(* Logix 5000 project; controller HP_SSC01 vendor 1 type 14 code 67 rev 17.7; software revision 17.01 *)

TASK MainTask (periodic, rate 10 ms, priority 5, watchdog 50 ms) : Main_SSC, Carousel1, Carousel2
TASK SafetyTask (periodic, rate 25 ms, priority 10, watchdog 20 ms) : Safe_SSC, SafeCarousel1

MODULES
   Local : vendor 1 type 14 code 67 (ICP 0, rev 17.7)
      SSC01_DNetSafeIO : vendor 1 type 12 code 14 (ICP 5, rev 10.5, Output RPI 20 ms, Input RPI 20 ms)
         SSC01_Safe2 : vendor 1 type 35 code 2 (DeviceNet 2, rev 1.2, Output RPI 25 ms, Input RPI 6 ms)
         C2_Safe : vendor 1 type 35 code 2 (DeviceNet 20, rev 1.2, Output RPI 25 ms, Input RPI 6 ms)
         SSC01_Safe3 : vendor 1 type 35 code 2 (DeviceNet 3, rev 1.2, Output RPI 25 ms, Input RPI 6 ms)
         C3_Safe : vendor 1 type 35 code 2 (DeviceNet 30, rev 1.2, Output RPI 25 ms, Input RPI 6 ms)
         SSC01_Safe1 : vendor 1 type 35 code 2 (DeviceNet 1, rev 1.2, Output RPI 25 ms, Input RPI 6 ms)
         C1_Safe : vendor 1 type 35 code 2 (DeviceNet 10, rev 1.2, Input RPI 6 ms, Output RPI 25 ms)
      HP_SSC01_0_3_ENBT : 1756-ENBT (ICP 3, Ethernet 192.168.201.51, rev 4.1)
         HP_RCS_RIDE_ENBT : 1756-ENBT (Ethernet 192.168.201.10, rev 4.1)
            @fd516503@:Partner : vendor 1 type 14 code 69 (ICP 1, rev 16.1)
            HP_RCS : vendor 1 type 14 code 67 (ICP 0, rev 16.1, $55e8e5d5$ RPI 25 ms)
      HP_SSC01_0_6_EN2T : 1756-EN2T (ICP 6, Ethernet 192.168.206.10, rev 1.3)
         C2_RIO_AENT : 1734-AENT (Ethernet 192.168.206.21, rev 2.3, Output RPI 20 ms)
            C2_RIO_1_IB8 : 1734-IB8 (PointIO 1, rev 3.1)
            C2_RIO_2_OB8 : 1734-OB8 (PointIO 2, rev 3.1)
            C2_RIO_3_SSI : vendor 1 type 115 code 80 (PointIO 3, rev 4.3, Output RPI 10 ms)
         C1_RIO_AENT : 1734-AENT (Ethernet 192.168.206.11, rev 2.3, Output RPI 20 ms)
            C1_RIO_1_IB8 : 1734-IB8 (PointIO 1, rev 3.1)
            C1_RIO_2_OB8 : 1734-OB8 (PointIO 2, rev 3.1)
            C1_RIO_3_SSI : vendor 1 type 115 code 80 (PointIO 3, rev 4.3, Output RPI 10 ms)
         C3_RIO_AENT : 1734-AENT (Ethernet 192.168.206.31, rev 2.3, Output RPI 20 ms)
            C3_RIO_1_IB8 : 1734-IB8 (PointIO 1, rev 3.1)
            C3_RIO_3_SSI : vendor 1 type 115 code 80 (PointIO 3, rev 4.3, Output RPI 10 ms)
            C3_RIO_2_OB8 : 1734-OB8 (PointIO 2, rev 3.1)
      HP_SSC01_0_2_ENBT : 1756-ENBT (ICP 2, Ethernet 192.168.202.11, rev 4.1)
      C1_SERCOS : vendor 1 type 16 code 13 (ICP 8, rev 17.1, MotionSync RPI 6 ms, MotionAsync RPI 25 ms, MotionEvent RPI 1000 ms)
         C1_K7K : vendor 1 type 115 code 182 (SERCOS 1, rev 1.1)
      C3_SERCOS : vendor 1 type 16 code 13 (ICP 10, rev 17.1, MotionSync RPI 6 ms, MotionAsync RPI 25 ms, MotionEvent RPI 1000 ms)
         C3_K7K : vendor 1 type 115 code 182 (SERCOS 3, rev 1.1)
      C2_SERCOS : vendor 1 type 16 code 13 (ICP 9, rev 17.1, MotionSync RPI 6 ms, MotionAsync RPI 25 ms, MotionEvent RPI 1000 ms)
         C2_K7K : vendor 1 type 115 code 182 (SERCOS 2, rev 1.1)
      @b5ff5b04@:Partner : vendor 1 type 14 code 69 (ICP 1, rev 17.7)
END_MODULES

TYPE FAULTRECORD :
STRUCT
   Time_Low : DINT;
   Time_High : DINT;
   Type : INT;
   Code : INT;
   Info : DINT[8];
END_STRUCT
END_TYPE

TYPE Profile_Table_Limits :
STRUCT
   On_Path_Low : REAL;
   On_Path_High : REAL;
   Near_On_Path_Low : REAL;
   Near_On_Path_High : REAL;
END_STRUCT
END_TYPE

TYPE UD_DTS :
STRUCT
   YEAR : DINT;
   MONTH : DINT;
   DAY : DINT;
   HOUR : DINT;
   MINUTE : DINT;
   SECOND : DINT;
   MIL_SEC : DINT;
END_STRUCT
END_TYPE

TYPE UD_FH_DATA :
STRUCT
   CODE : INT;
   MESSAGE : DINT;
   DATE_TIME : UD_DTS;
END_STRUCT
END_TYPE

TYPE UD_FH_LOG :
STRUCT
   MESSAGE : DINT;
   YEAR : DINT;
   MONTH : DINT;
   DAY : DINT;
   HOUR : DINT;
   MINUTE : DINT;
   SECOND : DINT;
   MIL_SEC : DINT;
END_STRUCT
END_TYPE

TYPE Udt_Carsl_SafeData :
STRUCT
   Status : CONNECTION_STATUS;
   Carsl_Status : DINT;
END_STRUCT
END_TYPE

TYPE Udt_Carsl_Stat :
STRUCT
   Enabled : BOOL;
   Mode : UDT_MODE;
   Posn : UDT_PositionProfile;
   Position : UDT_Parameter_Delta;
   CogNo : REAL;
   CogPosition : REAL;
   Velocity : REAL;
   PosnStatus : UDT_Position_Status;
   MotionCmdEn : BOOL;
   MotionActive : BOOL;
   realCog : REAL;
   realCogTot : REAL;
   RevCount : COUNTER;
   RevFlag : BOOL;
   Encoder_Secnd_Posn : REAL;
END_STRUCT
END_TYPE

TYPE UDT_Cog_Posn :
STRUCT
   CogNo : DINT;
   CogPosition : DINT;
   realCog : DINT;
   modCog : DINT;
END_STRUCT
END_TYPE

TYPE UDT_Encoder :
STRUCT
   Position : DINT;
   CntRaw : DINT;
   CntAdj : DINT;
   Initial : DINT;
   Delta : DINT;
   InitialPrev : DINT;
   CntMax : DINT;
   Rollover : DINT;
END_STRUCT
END_TYPE

TYPE UDT_GLX_ProduceConsume :
STRUCT
   Status : CONNECTION_STATUS;
   Data : DINT[5];
END_STRUCT
END_TYPE

TYPE UDT_MODE :
STRUCT
   Local : BOOL;
   Off : BOOL;
   Remote : BOOL;
   Unknown : BOOL;
END_STRUCT
END_TYPE

TYPE UDT_MOTION_STATE :
STRUCT
   Accel : BOOL;
   Run : BOOL;
   Decel : BOOL;
   Off : BOOL;
   OS : BOOL;
END_STRUCT
END_TYPE

TYPE UDT_Parameter_Delta :
STRUCT
   CurrentAbs : REAL;
   Initial : REAL;
   CurrentRel : REAL;
   Delta : REAL;
   Final : REAL;
END_STRUCT
END_TYPE

TYPE UDT_ParameterDint_Delta :
STRUCT
   Current : DINT;
   Initial : DINT;
   CurrentRel : DINT;
   Delta : DINT;
   Final : DINT;
END_STRUCT
END_TYPE

TYPE UDT_Position_Status :
STRUCT
   OnPath : BOOL;
   NearOnPath : BOOL;
   OffPath : BOOL;
   RecoveryZn : BOOL;
END_STRUCT
END_TYPE

TYPE UDT_PositionProfile :
STRUCT
   Initial : REAL;
   Accel : REAL;
   Stop : REAL;
   Final : REAL;
END_STRUCT
END_TYPE

TYPE Udt_RCS_SafeData :
STRUCT
   Status : CONNECTION_STATUS;
   Master_Clock : DINT;
   cst_Msec : DINT;
   cst_Sec : DINT;
   RailStateEthernet : DINT;
   Permissives : DINT;
END_STRUCT
END_TYPE

TYPE Udt_RCS_State :
STRUCT
   Value : DINT;
   Maint : BOOL;
   Add_Veh : BOOL;
   Second_Park : BOOL;
   Spare : BOOL;
   Stn_Park : BOOL;
   Reset_Flt : BOOL;
   Rem_Veh : BOOL;
   Go_Evac : BOOL;
   Inspect : BOOL;
   Inspect_Reset : BOOL;
   Retract_SAE : BOOL;
   Brake_Test : BOOL;
   Go_Keyhole : BOOL;
   Acq_MClock : BOOL;
   Go_MClock : BOOL;
   Inspect_Done : BOOL;
   StartUp_Keyhole : BOOL;
   Pri_Restart : BOOL;
   Stn_Evac : BOOL;
   Auto_Run : BOOL;
   Unknown : BOOL;
END_STRUCT
END_TYPE

TYPE UDT_Seqn :
STRUCT
   En : BOOL;
   OS : BOOL;
   Dn : BOOL;
   Flt : BOOL;
   Step : DINT;
   Tmr : TIMER;
END_STRUCT
END_TYPE

TYPE UDT_Test_Record :
STRUCT
   StartPosn : REAL;
   EndPosn : REAL;
   EndDist : REAL;
   TestTime : DINT;
   AccelPosn : REAL;
   AccelTime : DINT;
   AccelDist : REAL;
   AccelErrorHi : REAL;
   AccelErrorLo : REAL;
   RunPosn : REAL;
   RunTime : DINT;
   RunDist : REAL;
   RunErrorHi : REAL;
   RunErrorLo : REAL;
   DecelPosn : REAL;
   DecelTime : DINT;
   DecelDist : REAL;
   DecelErrorHi : REAL;
   DecelErrorLo : REAL;
END_STRUCT
END_TYPE

VAR_GLOBAL   (* controller tags *)
   A_C1_0200 : ALIAS FOR S_C1_FaultSafety.0;
   A_C1_0201 : ALIAS FOR S_C1_FaultSafety.1;
   A_C1_0202 : ALIAS FOR S_C1_FaultSafety.2;
   A_C1_0203 : ALIAS FOR S_C1_FaultSafety.3;
   A_C1_0204 : ALIAS FOR S_C1_FaultSafety.4;
   A_C1_0205 : ALIAS FOR S_C1_FaultSafety.5;
   A_C1_0206 : ALIAS FOR S_C1_FaultSafety.6;
   A_C1_0207 : ALIAS FOR S_C1_FaultSafety.7;
   A_C1_0208 : ALIAS FOR S_C1_FaultSafety.8;
   A_C1_0209 : ALIAS FOR S_C1_FaultSafety.9;
   A_C1_0210 : ALIAS FOR S_C1_FaultSafety.10;
   A_C1_0211 : ALIAS FOR S_C1_FaultSafety.11;
   A_C1_0212 : ALIAS FOR S_C1_FaultSafety.12;
   A_C1_0213 : ALIAS FOR S_C1_FaultSafety.13;
   A_C1_0214 : ALIAS FOR S_C1_FaultSafety.14;
   A_C1_0215 : ALIAS FOR S_C1_FaultSafety.15;
   A_C1_0216 : ALIAS FOR S_C1_FaultSafety.16;
   A_C1_0217 : ALIAS FOR S_C1_FaultSafety.17;
   A_C1_0218 : ALIAS FOR S_C1_FaultSafety.18;
   A_C1_0219 : ALIAS FOR S_C1_FaultSafety.19;
   A_C1_0220 : ALIAS FOR S_C1_FaultSafety.20;
   A_C1_0221 : ALIAS FOR S_C1_FaultSafety.21;
   A_C1_0222 : ALIAS FOR S_C1_FaultSafety.22;
   A_C1_0223 : ALIAS FOR S_C1_FaultSafety.23;
   A_C1_0224 : ALIAS FOR S_C1_FaultSafety.24;
   A_C1_0225 : ALIAS FOR S_C1_FaultSafety.25;
   A_C1_0226 : ALIAS FOR S_C1_FaultSafety.26;
   A_C1_0227 : ALIAS FOR S_C1_FaultSafety.27;
   A_C1_0228 : ALIAS FOR S_C1_FaultSafety.28;
   A_C1_0229 : ALIAS FOR S_C1_FaultSafety.29;
   A_C1_0230 : ALIAS FOR S_C1_FaultSafety.30;
   A_C1_0231 : ALIAS FOR S_C1_FaultSafety.31;
   A_C1_0300 : ALIAS FOR C1_FaultStandard.0;
   A_C1_0301 : ALIAS FOR C1_FaultStandard.1;
   A_C1_0302 : ALIAS FOR C1_FaultStandard.2;
   A_C1_0303 : ALIAS FOR C1_FaultStandard.3;
   A_C1_0304 : ALIAS FOR C1_FaultStandard.4;
   A_C1_0305 : ALIAS FOR C1_FaultStandard.5;
   A_C1_0306 : ALIAS FOR C1_FaultStandard.6;
   A_C1_0307 : ALIAS FOR C1_FaultStandard.7;
   A_C1_0308 : ALIAS FOR C1_FaultStandard.8;
   A_C1_0309 : ALIAS FOR C1_FaultStandard.9;
   A_C1_0310 : ALIAS FOR C1_FaultStandard.10;
   A_C1_0311 : ALIAS FOR C1_FaultStandard.11;
   A_C1_0312 : ALIAS FOR C1_FaultStandard.12;
   A_C1_0313 : ALIAS FOR C1_FaultStandard.13;
   A_C1_0314 : ALIAS FOR C1_FaultStandard.14;
   A_C1_0315 : ALIAS FOR C1_FaultStandard.15;
   A_C1_0316 : ALIAS FOR C1_FaultStandard.16;
   A_C1_0317 : ALIAS FOR C1_FaultStandard.17;
   A_C1_0318 : ALIAS FOR C1_FaultStandard.18;
   A_C1_0319 : ALIAS FOR C1_FaultStandard.19;
   A_C1_0320 : ALIAS FOR C1_FaultStandard.20;
   A_C1_0321 : ALIAS FOR C1_FaultStandard.21;
   A_C1_0322 : ALIAS FOR C1_FaultStandard.22;
   A_C1_0323 : ALIAS FOR C1_FaultStandard.23;
   A_C1_0324 : ALIAS FOR C1_FaultStandard.24;
   A_C1_0325 : ALIAS FOR C1_FaultStandard.25;
   A_C1_0326 : ALIAS FOR C1_FaultStandard.26;
   A_C1_0327 : ALIAS FOR C1_FaultStandard.27;
   A_C1_0328 : ALIAS FOR C1_FaultStandard.28;
   A_C1_0329 : ALIAS FOR C1_FaultStandard.29;
   A_C1_0330 : ALIAS FOR C1_FaultStandard.30;
   A_C1_0331 : ALIAS FOR C1_FaultStandard.31;
   A_C1_0400 : ALIAS FOR C1_Warning.0;
   A_C1_0401 : ALIAS FOR C1_Warning.1;
   A_C1_0402 : ALIAS FOR C1_Warning.2;
   A_C1_0403 : ALIAS FOR C1_Warning.3;
   A_C1_0404 : ALIAS FOR C1_Warning.4;
   A_C1_0405 : ALIAS FOR C1_Warning.5;
   A_C1_0406 : ALIAS FOR C1_Warning.6;
   A_C1_0407 : ALIAS FOR C1_Warning.7;
   A_C1_0408 : ALIAS FOR C1_Warning.8;
   A_C1_0409 : ALIAS FOR C1_Warning.9;
   A_C1_0410 : ALIAS FOR C1_Warning.10;
   A_C1_0411 : ALIAS FOR C1_Warning.11;
   A_C1_0412 : ALIAS FOR C1_Warning.12;
   A_C1_0413 : ALIAS FOR C1_Warning.13;
   A_C1_0414 : ALIAS FOR C1_Warning.14;
   A_C1_0415 : ALIAS FOR C1_Warning.15;
   A_C1_0416 : ALIAS FOR C1_Warning.16;
   A_C1_0417 : ALIAS FOR C1_Warning.17;
   A_C1_0418 : ALIAS FOR C1_Warning.18;
   A_C1_0419 : ALIAS FOR C1_Warning.19;
   A_C1_0420 : ALIAS FOR C1_Warning.20;
   A_C1_0421 : ALIAS FOR C1_Warning.21;
   A_C1_0422 : ALIAS FOR C1_Warning.22;
   A_C1_0423 : ALIAS FOR C1_Warning.23;
   A_C1_0424 : ALIAS FOR C1_Warning.24;
   A_C1_0425 : ALIAS FOR C1_Warning.25;
   A_C1_0426 : ALIAS FOR C1_Warning.26;
   A_C1_0427 : ALIAS FOR C1_Warning.27;
   A_C1_0428 : ALIAS FOR C1_Warning.28;
   A_C1_0429 : ALIAS FOR C1_Warning.29;
   A_C1_0430 : ALIAS FOR C1_Warning.30;
   A_C1_0431 : ALIAS FOR C1_Warning.31;
   A_C2_0200 : ALIAS FOR S_C2_FaultSafety.0;
   A_C2_0201 : ALIAS FOR S_C2_FaultSafety.1;
   A_C2_0202 : ALIAS FOR S_C2_FaultSafety.2;
   A_C2_0203 : ALIAS FOR S_C2_FaultSafety.3;
   A_C2_0204 : ALIAS FOR S_C2_FaultSafety.4;
   A_C2_0205 : ALIAS FOR S_C2_FaultSafety.5;
   A_C2_0206 : ALIAS FOR S_C2_FaultSafety.6;
   A_C2_0207 : ALIAS FOR S_C2_FaultSafety.7;
   A_C2_0208 : ALIAS FOR S_C2_FaultSafety.8;
   A_C2_0209 : ALIAS FOR S_C2_FaultSafety.9;
   A_C2_0210 : ALIAS FOR S_C2_FaultSafety.10;
   A_C2_0211 : ALIAS FOR S_C2_FaultSafety.11;
   A_C2_0212 : ALIAS FOR S_C2_FaultSafety.12;
   A_C2_0213 : ALIAS FOR S_C2_FaultSafety.13;
   A_C2_0214 : ALIAS FOR S_C2_FaultSafety.14;
   A_C2_0215 : ALIAS FOR S_C2_FaultSafety.15;
   A_C2_0216 : ALIAS FOR S_C2_FaultSafety.16;
   A_C2_0217 : ALIAS FOR S_C2_FaultSafety.17;
   A_C2_0218 : ALIAS FOR S_C2_FaultSafety.18;
   A_C2_0219 : ALIAS FOR S_C2_FaultSafety.19;
   A_C2_0220 : ALIAS FOR S_C2_FaultSafety.20;
   A_C2_0221 : ALIAS FOR S_C2_FaultSafety.21;
   A_C2_0222 : ALIAS FOR S_C2_FaultSafety.22;
   A_C2_0223 : ALIAS FOR S_C2_FaultSafety.23;
   A_C2_0224 : ALIAS FOR S_C2_FaultSafety.24;
   A_C2_0225 : ALIAS FOR S_C2_FaultSafety.25;
   A_C2_0226 : ALIAS FOR S_C2_FaultSafety.26;
   A_C2_0227 : ALIAS FOR S_C2_FaultSafety.27;
   A_C2_0228 : ALIAS FOR S_C2_FaultSafety.28;
   A_C2_0229 : ALIAS FOR S_C2_FaultSafety.29;
   A_C2_0230 : ALIAS FOR S_C2_FaultSafety.30;
   A_C2_0231 : ALIAS FOR S_C2_FaultSafety.31;
   A_C2_0300 : ALIAS FOR C2_FaultStandard.0;
   A_C2_0301 : ALIAS FOR C2_FaultStandard.1;
   A_C2_0302 : ALIAS FOR C2_FaultStandard.2;
   A_C2_0303 : ALIAS FOR C2_FaultStandard.3;
   A_C2_0304 : ALIAS FOR C2_FaultStandard.4;
   A_C2_0305 : ALIAS FOR C2_FaultStandard.5;
   A_C2_0306 : ALIAS FOR C2_FaultStandard.6;
   A_C2_0307 : ALIAS FOR C2_FaultStandard.7;
   A_C2_0308 : ALIAS FOR C2_FaultStandard.8;
   A_C2_0309 : ALIAS FOR C2_FaultStandard.9;
   A_C2_0310 : ALIAS FOR C2_FaultStandard.10;
   A_C2_0311 : ALIAS FOR C2_FaultStandard.11;
   A_C2_0312 : ALIAS FOR C2_FaultStandard.12;
   A_C2_0313 : ALIAS FOR C2_FaultStandard.13;
   A_C2_0314 : ALIAS FOR C2_FaultStandard.14;
   A_C2_0315 : ALIAS FOR C2_FaultStandard.15;
   A_C2_0316 : ALIAS FOR C2_FaultStandard.16;
   A_C2_0317 : ALIAS FOR C2_FaultStandard.17;
   A_C2_0318 : ALIAS FOR C2_FaultStandard.18;
   A_C2_0319 : ALIAS FOR C2_FaultStandard.19;
   A_C2_0320 : ALIAS FOR C2_FaultStandard.20;
   A_C2_0321 : ALIAS FOR C2_FaultStandard.21;
   A_C2_0322 : ALIAS FOR C2_FaultStandard.22;
   A_C2_0323 : ALIAS FOR C2_FaultStandard.23;
   A_C2_0324 : ALIAS FOR C2_FaultStandard.24;
   A_C2_0325 : ALIAS FOR C2_FaultStandard.25;
   A_C2_0326 : ALIAS FOR C2_FaultStandard.26;
   A_C2_0327 : ALIAS FOR C2_FaultStandard.27;
   A_C2_0328 : ALIAS FOR C2_FaultStandard.28;
   A_C2_0329 : ALIAS FOR C2_FaultStandard.29;
   A_C2_0330 : ALIAS FOR C2_FaultStandard.30;
   A_C2_0331 : ALIAS FOR C2_FaultStandard.31;
   A_C2_0400 : ALIAS FOR C2_Warning.0;
   A_C2_0401 : ALIAS FOR C2_Warning.1;
   A_C2_0402 : ALIAS FOR C2_Warning.2;
   A_C2_0403 : ALIAS FOR C2_Warning.3;
   A_C2_0404 : ALIAS FOR C2_Warning.4;
   A_C2_0405 : ALIAS FOR C2_Warning.5;
   A_C2_0406 : ALIAS FOR C2_Warning.6;
   A_C2_0407 : ALIAS FOR C2_Warning.7;
   A_C2_0408 : ALIAS FOR C2_Warning.8;
   A_C2_0409 : ALIAS FOR C2_Warning.9;
   A_C2_0410 : ALIAS FOR C2_Warning.10;
   A_C2_0411 : ALIAS FOR C2_Warning.11;
   A_C2_0412 : ALIAS FOR C2_Warning.12;
   A_C2_0413 : ALIAS FOR C2_Warning.13;
   A_C2_0414 : ALIAS FOR C2_Warning.14;
   A_C2_0415 : ALIAS FOR C2_Warning.15;
   A_C2_0416 : ALIAS FOR C2_Warning.16;
   A_C2_0417 : ALIAS FOR C2_Warning.17;
   A_C2_0418 : ALIAS FOR C2_Warning.18;
   A_C2_0419 : ALIAS FOR C2_Warning.19;
   A_C2_0420 : ALIAS FOR C2_Warning.20;
   A_C2_0421 : ALIAS FOR C2_Warning.21;
   A_C2_0422 : ALIAS FOR C2_Warning.22;
   A_C2_0423 : ALIAS FOR C2_Warning.23;
   A_C2_0424 : ALIAS FOR C2_Warning.24;
   A_C2_0425 : ALIAS FOR C2_Warning.25;
   A_C2_0426 : ALIAS FOR C2_Warning.26;
   A_C2_0427 : ALIAS FOR C2_Warning.27;
   A_C2_0428 : ALIAS FOR C2_Warning.28;
   A_C2_0429 : ALIAS FOR C2_Warning.29;
   A_C2_0430 : ALIAS FOR C2_Warning.30;
   A_C2_0431 : ALIAS FOR C2_Warning.31;
   A_C3_0200 : ALIAS FOR S_C3_FaultSafety.0;
   A_C3_0201 : ALIAS FOR S_C3_FaultSafety.1;
   A_C3_0202 : ALIAS FOR S_C3_FaultSafety.2;
   A_C3_0203 : ALIAS FOR S_C3_FaultSafety.3;
   A_C3_0204 : ALIAS FOR S_C3_FaultSafety.4;
   A_C3_0205 : ALIAS FOR S_C3_FaultSafety.5;
   A_C3_0206 : ALIAS FOR S_C3_FaultSafety.6;
   A_C3_0207 : ALIAS FOR S_C3_FaultSafety.7;
   A_C3_0208 : ALIAS FOR S_C3_FaultSafety.8;
   A_C3_0209 : ALIAS FOR S_C3_FaultSafety.9;
   A_C3_0210 : ALIAS FOR S_C3_FaultSafety.10;
   A_C3_0211 : ALIAS FOR S_C3_FaultSafety.11;
   A_C3_0212 : ALIAS FOR S_C3_FaultSafety.12;
   A_C3_0213 : ALIAS FOR S_C3_FaultSafety.13;
   A_C3_0214 : ALIAS FOR S_C3_FaultSafety.14;
   A_C3_0215 : ALIAS FOR S_C3_FaultSafety.15;
   A_C3_0216 : ALIAS FOR S_C3_FaultSafety.16;
   A_C3_0217 : ALIAS FOR S_C3_FaultSafety.17;
   A_C3_0218 : ALIAS FOR S_C3_FaultSafety.18;
   A_C3_0219 : ALIAS FOR S_C3_FaultSafety.19;
   A_C3_0220 : ALIAS FOR S_C3_FaultSafety.20;
   A_C3_0221 : ALIAS FOR S_C3_FaultSafety.21;
   A_C3_0222 : ALIAS FOR S_C3_FaultSafety.22;
   A_C3_0223 : ALIAS FOR S_C3_FaultSafety.23;
   A_C3_0224 : ALIAS FOR S_C3_FaultSafety.24;
   A_C3_0225 : ALIAS FOR S_C3_FaultSafety.25;
   A_C3_0226 : ALIAS FOR S_C3_FaultSafety.26;
   A_C3_0227 : ALIAS FOR S_C3_FaultSafety.27;
   A_C3_0228 : ALIAS FOR S_C3_FaultSafety.28;
   A_C3_0229 : ALIAS FOR S_C3_FaultSafety.29;
   A_C3_0230 : ALIAS FOR S_C3_FaultSafety.30;
   A_C3_0231 : ALIAS FOR S_C3_FaultSafety.31;
   A_C3_0300 : ALIAS FOR C3_FaultStandard.0;
   A_C3_0301 : ALIAS FOR C3_FaultStandard.1;
   A_C3_0302 : ALIAS FOR C3_FaultStandard.2;
   A_C3_0303 : ALIAS FOR C3_FaultStandard.3;
   A_C3_0304 : ALIAS FOR C3_FaultStandard.4;
   A_C3_0305 : ALIAS FOR C3_FaultStandard.5;
   A_C3_0306 : ALIAS FOR C3_FaultStandard.6;
   A_C3_0307 : ALIAS FOR C3_FaultStandard.7;
   A_C3_0308 : ALIAS FOR C3_FaultStandard.8;
   A_C3_0309 : ALIAS FOR C3_FaultStandard.9;
   A_C3_0310 : ALIAS FOR C3_FaultStandard.10;
   A_C3_0311 : ALIAS FOR C3_FaultStandard.11;
   A_C3_0312 : ALIAS FOR C3_FaultStandard.12;
   A_C3_0313 : ALIAS FOR C3_FaultStandard.13;
   A_C3_0314 : ALIAS FOR C3_FaultStandard.14;
   A_C3_0315 : ALIAS FOR C3_FaultStandard.15;
   A_C3_0316 : ALIAS FOR C3_FaultStandard.16;
   A_C3_0317 : ALIAS FOR C3_FaultStandard.17;
   A_C3_0318 : ALIAS FOR C3_FaultStandard.18;
   A_C3_0319 : ALIAS FOR C3_FaultStandard.19;
   A_C3_0320 : ALIAS FOR C3_FaultStandard.20;
   A_C3_0321 : ALIAS FOR C3_FaultStandard.21;
   A_C3_0322 : ALIAS FOR C3_FaultStandard.22;
   A_C3_0323 : ALIAS FOR C3_FaultStandard.23;
   A_C3_0324 : ALIAS FOR C3_FaultStandard.24;
   A_C3_0325 : ALIAS FOR C3_FaultStandard.25;
   A_C3_0326 : ALIAS FOR C3_FaultStandard.26;
   A_C3_0327 : ALIAS FOR C3_FaultStandard.27;
   A_C3_0328 : ALIAS FOR C3_FaultStandard.28;
   A_C3_0329 : ALIAS FOR C3_FaultStandard.29;
   A_C3_0330 : ALIAS FOR C3_FaultStandard.30;
   A_C3_0331 : ALIAS FOR C3_FaultStandard.31;
   A_C3_0400 : ALIAS FOR C3_Warning.0;
   A_C3_0401 : ALIAS FOR C3_Warning.1;
   A_C3_0402 : ALIAS FOR C3_Warning.2;
   A_C3_0403 : ALIAS FOR C3_Warning.3;
   A_C3_0404 : ALIAS FOR C3_Warning.4;
   A_C3_0405 : ALIAS FOR C3_Warning.5;
   A_C3_0406 : ALIAS FOR C3_Warning.6;
   A_C3_0407 : ALIAS FOR C3_Warning.7;
   A_C3_0408 : ALIAS FOR C3_Warning.8;
   A_C3_0409 : ALIAS FOR C3_Warning.9;
   A_C3_0410 : ALIAS FOR C3_Warning.10;
   A_C3_0411 : ALIAS FOR C3_Warning.11;
   A_C3_0412 : ALIAS FOR C3_Warning.12;
   A_C3_0413 : ALIAS FOR C3_Warning.13;
   A_C3_0414 : ALIAS FOR C3_Warning.14;
   A_C3_0415 : ALIAS FOR C3_Warning.15;
   A_C3_0416 : ALIAS FOR C3_Warning.16;
   A_C3_0417 : ALIAS FOR C3_Warning.17;
   A_C3_0418 : ALIAS FOR C3_Warning.18;
   A_C3_0419 : ALIAS FOR C3_Warning.19;
   A_C3_0420 : ALIAS FOR C3_Warning.20;
   A_C3_0421 : ALIAS FOR C3_Warning.21;
   A_C3_0422 : ALIAS FOR C3_Warning.22;
   A_C3_0423 : ALIAS FOR C3_Warning.23;
   A_C3_0424 : ALIAS FOR C3_Warning.24;
   A_C3_0425 : ALIAS FOR C3_Warning.25;
   A_C3_0426 : ALIAS FOR C3_Warning.26;
   A_C3_0427 : ALIAS FOR C3_Warning.27;
   A_C3_0428 : ALIAS FOR C3_Warning.28;
   A_C3_0429 : ALIAS FOR C3_Warning.29;
   A_C3_0430 : ALIAS FOR C3_Warning.30;
   A_C3_0431 : ALIAS FOR C3_Warning.31;
   A_S01_0100 : ALIAS FOR System_FaultSafeIO.0;
   A_S01_0101 : ALIAS FOR System_FaultSafeIO.1;
   A_S01_0102 : ALIAS FOR System_FaultSafeIO.2;
   A_S01_0103 : ALIAS FOR System_FaultSafeIO.3;
   A_S01_0104 : ALIAS FOR System_FaultSafeIO.4;
   A_S01_0105 : ALIAS FOR System_FaultSafeIO.5;
   A_S01_0106 : ALIAS FOR System_FaultSafeIO.6;
   A_S01_0107 : ALIAS FOR System_FaultSafeIO.7;
   A_S01_0108 : ALIAS FOR System_FaultSafeIO.8;
   A_S01_0109 : ALIAS FOR System_FaultSafeIO.9;
   A_S01_0110 : ALIAS FOR System_FaultSafeIO.10;
   A_S01_0111 : ALIAS FOR System_FaultSafeIO.11;
   A_S01_0112 : ALIAS FOR System_FaultSafeIO.12;
   A_S01_0113 : ALIAS FOR System_FaultSafeIO.13;
   A_S01_0114 : ALIAS FOR System_FaultSafeIO.14;
   A_S01_0115 : ALIAS FOR System_FaultSafeIO.15;
   A_S01_0116 : ALIAS FOR System_FaultSafeIO.16;
   A_S01_0117 : ALIAS FOR System_FaultSafeIO.17;
   A_S01_0118 : ALIAS FOR System_FaultSafeIO.18;
   A_S01_0119 : ALIAS FOR System_FaultSafeIO.19;
   A_S01_0120 : ALIAS FOR System_FaultSafeIO.20;
   A_S01_0121 : ALIAS FOR System_FaultSafeIO.21;
   A_S01_0122 : ALIAS FOR System_FaultSafeIO.22;
   A_S01_0123 : ALIAS FOR System_FaultSafeIO.23;
   A_S01_0124 : ALIAS FOR System_FaultSafeIO.24;
   A_S01_0125 : ALIAS FOR System_FaultSafeIO.25;
   A_S01_0126 : ALIAS FOR System_FaultSafeIO.26;
   A_S01_0127 : ALIAS FOR System_FaultSafeIO.27;
   A_S01_0128 : ALIAS FOR System_FaultSafeIO.28;
   A_S01_0129 : ALIAS FOR System_FaultSafeIO.29;
   A_S01_0130 : ALIAS FOR System_FaultSafeIO.30;
   A_S01_0131 : ALIAS FOR System_FaultSafeIO.31;
   A_S01_0200 : ALIAS FOR System_FaultSafety.0;
   A_S01_0201 : ALIAS FOR System_FaultSafety.1;
   A_S01_0202 : ALIAS FOR System_FaultSafety.2;
   A_S01_0203 : ALIAS FOR System_FaultSafety.3;
   A_S01_0204 : ALIAS FOR System_FaultSafety.4;
   A_S01_0205 : ALIAS FOR System_FaultSafety.5;
   A_S01_0206 : ALIAS FOR System_FaultSafety.6;
   A_S01_0207 : ALIAS FOR System_FaultSafety.7;
   A_S01_0208 : ALIAS FOR System_FaultSafety.8;
   A_S01_0209 : ALIAS FOR System_FaultSafety.9;
   A_S01_0210 : ALIAS FOR System_FaultSafety.10;
   A_S01_0211 : ALIAS FOR System_FaultSafety.11;
   A_S01_0212 : ALIAS FOR System_FaultSafety.12;
   A_S01_0213 : ALIAS FOR System_FaultSafety.13;
   A_S01_0214 : ALIAS FOR System_FaultSafety.14;
   A_S01_0215 : ALIAS FOR System_FaultSafety.15;
   A_S01_0216 : ALIAS FOR System_FaultSafety.16;
   A_S01_0217 : ALIAS FOR System_FaultSafety.17;
   A_S01_0218 : ALIAS FOR System_FaultSafety.18;
   A_S01_0219 : ALIAS FOR System_FaultSafety.19;
   A_S01_0220 : ALIAS FOR System_FaultSafety.20;
   A_S01_0221 : ALIAS FOR System_FaultSafety.21;
   A_S01_0222 : ALIAS FOR System_FaultSafety.22;
   A_S01_0223 : ALIAS FOR System_FaultSafety.23;
   A_S01_0224 : ALIAS FOR System_FaultSafety.24;
   A_S01_0225 : ALIAS FOR System_FaultSafety.25;
   A_S01_0226 : ALIAS FOR System_FaultSafety.26;
   A_S01_0227 : ALIAS FOR System_FaultSafety.27;
   A_S01_0228 : ALIAS FOR System_FaultSafety.28;
   A_S01_0229 : ALIAS FOR System_FaultSafety.29;
   A_S01_0230 : ALIAS FOR System_FaultSafety.30;
   A_S01_0231 : ALIAS FOR System_FaultSafety.31;
   A_S01_0300 : ALIAS FOR System_FaultStandard.0;
   A_S01_0301 : ALIAS FOR System_FaultStandard.1;
   A_S01_0302 : ALIAS FOR System_FaultStandard.2;
   A_S01_0303 : ALIAS FOR System_FaultStandard.3;
   A_S01_0304 : ALIAS FOR System_FaultStandard.4;
   A_S01_0305 : ALIAS FOR System_FaultStandard.5;
   A_S01_0306 : ALIAS FOR System_FaultStandard.6;
   A_S01_0307 : ALIAS FOR System_FaultStandard.7;
   A_S01_0308 : ALIAS FOR System_FaultStandard.8;
   A_S01_0309 : ALIAS FOR System_FaultStandard.9;
   A_S01_0310 : ALIAS FOR System_FaultStandard.10;
   A_S01_0311 : ALIAS FOR System_FaultStandard.11;
   A_S01_0312 : ALIAS FOR System_FaultStandard.12;
   A_S01_0313 : ALIAS FOR System_FaultStandard.13;
   A_S01_0314 : ALIAS FOR System_FaultStandard.14;
   A_S01_0315 : ALIAS FOR System_FaultStandard.15;
   A_S01_0316 : ALIAS FOR System_FaultStandard.16;
   A_S01_0317 : ALIAS FOR System_FaultStandard.17;
   A_S01_0318 : ALIAS FOR System_FaultStandard.18;
   A_S01_0319 : ALIAS FOR System_FaultStandard.19;
   A_S01_0320 : ALIAS FOR System_FaultStandard.20;
   A_S01_0321 : ALIAS FOR System_FaultStandard.21;
   A_S01_0322 : ALIAS FOR System_FaultStandard.22;
   A_S01_0323 : ALIAS FOR System_FaultStandard.23;
   A_S01_0324 : ALIAS FOR System_FaultStandard.24;
   A_S01_0325 : ALIAS FOR System_FaultStandard.25;
   A_S01_0326 : ALIAS FOR System_FaultStandard.26;
   A_S01_0327 : ALIAS FOR System_FaultStandard.27;
   A_S01_0328 : ALIAS FOR System_FaultStandard.28;
   A_S01_0329 : ALIAS FOR System_FaultStandard.29;
   A_S01_0330 : ALIAS FOR System_FaultStandard.30;
   A_S01_0331 : ALIAS FOR System_FaultStandard.31;
   A_S01_0400 : ALIAS FOR System_Warning.0;
   A_S01_0401 : ALIAS FOR System_Warning.1;
   A_S01_0402 : ALIAS FOR System_Warning.2;
   A_S01_0403 : ALIAS FOR System_Warning.3;
   A_S01_0404 : ALIAS FOR System_Warning.4;
   A_S01_0405 : ALIAS FOR System_Warning.5;
   A_S01_0406 : ALIAS FOR System_Warning.6;
   A_S01_0407 : ALIAS FOR System_Warning.7;
   A_S01_0408 : ALIAS FOR System_Warning.8;
   A_S01_0409 : ALIAS FOR System_Warning.9;
   A_S01_0410 : ALIAS FOR System_Warning.10;
   A_S01_0411 : ALIAS FOR System_Warning.11;
   A_S01_0412 : ALIAS FOR System_Warning.12;
   A_S01_0413 : ALIAS FOR System_Warning.13;
   A_S01_0414 : ALIAS FOR System_Warning.14;
   A_S01_0415 : ALIAS FOR System_Warning.15;
   A_S01_0416 : ALIAS FOR System_Warning.16;
   A_S01_0417 : ALIAS FOR System_Warning.17;
   A_S01_0418 : ALIAS FOR System_Warning.18;
   A_S01_0419 : ALIAS FOR System_Warning.19;
   A_S01_0420 : ALIAS FOR System_Warning.20;
   A_S01_0421 : ALIAS FOR System_Warning.21;
   A_S01_0422 : ALIAS FOR System_Warning.22;
   A_S01_0423 : ALIAS FOR System_Warning.23;
   A_S01_0424 : ALIAS FOR System_Warning.24;
   A_S01_0425 : ALIAS FOR System_Warning.25;
   A_S01_0426 : ALIAS FOR System_Warning.26;
   A_S01_0427 : ALIAS FOR System_Warning.27;
   A_S01_0428 : ALIAS FOR System_Warning.28;
   A_S01_0429 : ALIAS FOR System_Warning.29;
   A_S01_0430 : ALIAS FOR System_Warning.30;
   A_S01_0431 : ALIAS FOR System_Warning.31;
   Bit : BOOL;
   C01_SafeMemory : Udt_Carsl_SafeData := (Carsl_Status := 285); {produced}
   C02_SafeMemory : Udt_Carsl_SafeData := (Carsl_Status := 261); {produced}
   C03_SafeMemory : Udt_Carsl_SafeData := (Carsl_Status := 285); {produced}
   C1 : AXIS_SERVO_DRIVE;
   C1_32HourTimers : TIMER[8] := ([0].PRE := 115200000, [1].PRE := 115200000, [1].ACC := 1310840, [1].EN := 1, [1].TT := 1, [2].PRE := 115200000, [2].ACC := 11902210, [2].EN := 1, [2].TT := 1, [3].PRE := 115200000);
   C1_ActualPositionMOD60 : REAL := 41.785645;
   C1_All_DLY_OK : BOOL;
   C1_Brake_Daily_ok : BOOL;
   C1_Brake_Test_passed : BOOL := 1;
   C1_BrakeReleaseSelected : BOOL;
   C1_BrakeSequenceInProcess : BOOL;
   C1_BrakeTest : BOOL;
   C1_BrakeTestEndPosition : REAL := 3.4107273;
   C1_BrakeTestExpireTime : DINT := 32;
   C1_BrakeTestExpireTimeTemp : DINT := 115200000;
   C1_BrakeTestFailed : BOOL;
   C1_BrakeTestLocalDisable : BOOL;
   C1_BrakeTestMAJ01 : MOTION_INSTRUCTION := (FLAGS := 33554432);
   C1_BrakeTestMessageNumber : DINT;
   C1_BrakeTestONS : BOOL;
   C1_BrakeTestSelected : BOOL;
   C1_BrakeTestSequence : DINT;
   C1_BrakeTestSequenceAlarms : DINT;
   C1_BrakeTestSequenceAlarmTimer : TIMER[16] := ([0].PRE := 300000, [1].PRE := 30000000, [2].PRE := 300000, [3].PRE := 300000, [4].PRE := 300000, [5].PRE := 300000, [6].PRE := 300000, [7].PRE := 300000, [8].PRE := 300000, [9].PRE := 300000, [10].PRE := 300000);
   C1_BrakeTestSequenceONS : DINT;
   C1_BrakeTestStartPosition : REAL := 1.1649486;
   C1_BrakeTestStoppingDistance : REAL := 2.2457786;
   C1_BrakeTestTimerHoldVel : TIMER := (PRE := 1000);
   C1_BrakeTestWarning : BOOL;
   C1_DisableTimer : TIMER := (PRE := 1000);
   C1_DistanceToEvac : REAL := 7.999359;
   C1_Dump_OK : BOOL;
   C1_DumpTest : BOOL;
   C1_DumpValveFailedOff : BOOL;
   C1_DumpValveFailedOn : BOOL;
   C1_DumpValveMessageNumber : DINT;
   C1_DumpValveReleaseSelected : BOOL;
   C1_DumpValveTestDelay : TIMER[4] := ([0].PRE := 10000, [1].PRE := 10000, [2].PRE := 5000, [3].PRE := 5000);
   C1_DumpValveTestDelay2 : TIMER := (PRE := 5000);
   C1_DumpValveTestExpireTime : DINT := 32;
   C1_DumpValveTestExpireTimeTemp : DINT := 115200000;
   C1_DumpValveTestSelected : BOOL;
   C1_DumpValveTestSequence : DINT;
   C1_DumpValveTestSequenceAlarms : DINT;
   C1_DumpValveTestSequenceAlarmTimer : TIMER[16] := ([0].PRE := 300000, [1].PRE := 300000, [2].PRE := 300000, [3].PRE := 300000, [4].PRE := 300000, [5].PRE := 300000, [6].PRE := 300000, [7].PRE := 300000, [8].PRE := 300000, [9].PRE := 300000, [10].PRE := 300000);
   C1_EncoderCounts : DINT := 819093;
   C1_EncoderCountsRaw : ALIAS FOR C1_RIO_AENT:3:I.PresentData;
   C1_EncoderDegree : REAL := 341.712;
   C1_EncoderPositionAtHome : DINT := 4345814;
   C1_Error_Message_Raw : SINT[82] := ([0] := 64, [4] := 80, [5] := 104, [6] := 97, [7] := 115, [8] := 101, [9] := 32, [10] := 76, [11] := 111, [12] := 115, [13] := 115, [14] := 32, [15] := 70, [16] := 108, [17] := 116, [18] := 32, [19] := 32, [20] := 32);
   C1_EvacInPositionTest : DINT := 49785;
   C1_EvacPosition : REAL := 349.785;
   C1_EvacPositionMOD60 : REAL := 49.785004;
   C1_ExcecutePBHoldTimer : TIMER := (PRE := 5000);
   C1_FaultDebounce : TIMER[16] := ([0].PRE := 1250, [1].PRE := 500, [1].ACC := 500, [1].EN := 1, [1].DN := 1, [2].PRE := 1500, [3].PRE := 250, [4].PRE := 20);
   C1_FaultHoldTimer : TIMER[8] := ([0].PRE := 5000, [1].PRE := 5000);
   C1_FaultHomeSwitchNotFound : BOOL;
   C1_FaultStandard : DINT;
   C1_GoNearOnPathDelay : TIMER := (PRE := 2000);
   C1_GoToEvacMAM01 : MOTION_INSTRUCTION := (FLAGS := 33554432);
   C1_GoToOnPathMAM01 : MOTION_INSTRUCTION := (FLAGS := 704643072, DN := 1, PC := 1);
   C1_GoToOnPathMAM02 : MOTION_INSTRUCTION := (FLAGS := 33554432);
   C1_Home_OK : BOOL := 1;
   C1_Homed : BOOL := 1;
   C1_HomeDelay : TIMER[16] := ([0].PRE := 2000, [1].PRE := 2000, [2].PRE := 4000, [3].PRE := 2000, [4].PRE := 2000, [5].PRE := 1000, [6].PRE := 1000, [7].PRE := 3000);
   C1_HomeExpireTime : DINT := 31;
   C1_HomeExpireTimeTemp : DINT := 113890210;
   C1_HomeFindSwitchMAM01 : MOTION_INSTRUCTION := (FLAGS := 570425344, DN := 1);
   C1_HomeFindSwitchMAM02 : MOTION_INSTRUCTION := (FLAGS := 704643072, DN := 1, PC := 1);
   C1_HomeFindSwitchMAS01 : MOTION_INSTRUCTION := (FLAGS := 704643072, DN := 1, PC := 1);
   C1_HomeGetCloseToSwitchMAM01 : MOTION_INSTRUCTION := (FLAGS := 33554432);
   C1_HomeGoToOnPathMAM01 : MOTION_INSTRUCTION := (FLAGS := 704643072, DN := 1, PC := 1);
   C1_HomeInputStatus : BOOL := 1;
   C1_HomeMessageNumber : DINT := -2147483648;
   C1_HomeSensorTestMAM02 : MOTION_INSTRUCTION := (FLAGS := 704643072, DN := 1, PC := 1);
   C1_HomeSequence : DINT := -2147483648;
   C1_HomeSequenceAlarms : DINT;
   C1_HomeSequenceAlarmTimer : TIMER[32] := ([0].PRE := 300000, [1].PRE := 300000, [2].PRE := 300000, [3].PRE := 300000, [4].PRE := 300000, [5].PRE := 300000, [6].PRE := 300000, [7].PRE := 300000, [8].PRE := 300000, [9].PRE := 300000, [10].PRE := 300000, [11].PRE := 300000, [12].PRE := 300000, [13].PRE := 300000, [14].PRE := 300000, [15].PRE := 300000, [16].PRE := 300000, [17].PRE := 300000, [18].PRE := 300000, [19].PRE := 300000, [20].PRE := 300000, [21].PRE := 300000, [22].PRE := 300000);
   C1_HomeSequenceInProcess : BOOL;
   C1_HomeSequenceMAH : MOTION_INSTRUCTION := (FLAGS := 671088640, DN := 1, PC := 1, STATE := 17);
   C1_HomeSwitchFaultK7KFailedOff : BOOL;
   C1_HomeSwitchFaultK7KFailedOn : BOOL;
   C1_HomeSwitchFaultSafeFailedOff : BOOL;
   C1_HomeSwitchFaultSafeFailedOn : BOOL;
   C1_HomeTest : REAL := 248.31882;
   C1_IndexEnable : BOOL;
   C1_IndexEnableTOF : TIMER := (PRE := 5000, ACC := 5000);
   C1_IndexMAM01 : MOTION_INSTRUCTION := (FLAGS := 33554432);
   C1_IndexMAS01 : MOTION_INSTRUCTION := (FLAGS := 33554432);
   C1_IndexMessageNumber : DINT;
   C1_IndexPermissive : BOOL;
   C1_Jog_ONS : DINT;
   C1_JogDirection : DINT := 1;
   C1_JogEnable : BOOL;
   C1_JogEnableTOF : TIMER := (PRE := 15000, ACC := 15000);
   C1_JogForwardFastSelected : BOOL;
   C1_JogForwardSlowSelected : BOOL;
   C1_JogMAJ01 : MOTION_INSTRUCTION := (FLAGS := 570425344, DN := 1);
   C1_JogMAJ02 : MOTION_INSTRUCTION := (FLAGS := 33554432);
   C1_JogMAS01 : MOTION_INSTRUCTION := (FLAGS := 704643072, DN := 1, PC := 1);
   C1_JogMessageNumber : DINT;
   C1_JogPermissive : BOOL;
   C1_JogReverseFastSelected : BOOL;
   C1_JogReverseSlowSelected : BOOL;
   C1_LIM_ALARM_B : ALIAS FOR C1_RIO_AENT:I.Data[1].0;
   C1_LubricationMessageNumber : DINT;
   C1_LubricationOnTimer : TIMER := (PRE := 5000);
   C1_LubricationOverrideSelected : BOOL;
   C1_MAFR : MOTION_INSTRUCTION := (FLAGS := 301989888, ER := 1, ERR := 11);
   C1_MAG : MOTION_INSTRUCTION := (FLAGS := 33554432);
   C1_MaintEnable : BOOL;
   C1_MAJAcceleration : REAL := 3.0;
   C1_MAJDeceleration : REAL := 5.0;
   C1_MAJSpeed : REAL := 8.5714;
   C1_MAS : MOTION_INSTRUCTION := (FLAGS := 33554432);
   C1_MASR : MOTION_INSTRUCTION := (FLAGS := 33554432);
   C1_MotorActualPositionX1000 : DINT := 341786;
   C1_MotorAverageVelocityX1000 : DINT;
   C1_MotorFan : ALIAS FOR C1_RIO_AENT:O.Data[2].0;
   C1_MSF : MOTION_INSTRUCTION := (FLAGS := 536870912, DN := 1, STATUS := 2, STATE := 1);
   C1_MSO : MOTION_INSTRUCTION := (FLAGS := 536870912, DN := 1, STATE := 1);
   C1_Oiler : ALIAS FOR C1_RIO_AENT:O.Data[2].1;
   C1_OIT_BrakeRelease : BOOL;
   C1_OIT_BrakeReleaseDisplay : BOOL;
   C1_OIT_BrakeTest : BOOL;
   C1_OIT_BrakeTestDisplay : BOOL;
   C1_OIT_Command : DINT := 20;
   C1_OIT_Current : DINT := 20;
   C1_OIT_DumpValveRelease : BOOL;
   C1_OIT_DumpValveReleaseDisplay : BOOL;
   C1_OIT_DumpValveTest : BOOL;
   C1_OIT_DumpValveTestDisplay : BOOL;
   C1_OIT_FaultReset : BOOL;
   C1_OIT_FaultsExist : BOOL;
   C1_OIT_HomeCountDown : DINT := 6;
   C1_OIT_JogForwardFast : BOOL;
   C1_OIT_JogForwardFastDisplay : BOOL;
   C1_OIT_JogForwardSlow : BOOL;
   C1_OIT_JogForwardSlowDisplay : BOOL;
   C1_OIT_JogReverseFast : BOOL;
   C1_OIT_JogReverseFastDisplay : BOOL;
   C1_OIT_JogReverseSlow : BOOL;
   C1_OIT_JogReverseSlowDisplay : BOOL;
   C1_OIT_JogStopDisplay : BOOL := 1;
   C1_OIT_LubricationOverride : BOOL;
   C1_OIT_LubricationOverrideDisplay : BOOL;
   C1_OIT_PathError : DINT := -2077;
   C1_OIT_PathIndicatorHigh : DINT := 546;
   C1_OIT_PathIndicatorLow : DINT := -546;
   C1_OIT_WarningsExist : BOOL := 1;
   C1_OneTryToFixErrorONS : BOOL;
   C1_ONS : DINT;
   C1_ONS_Fault : DINT;
   C1_RemoteBrakeAndHomeSequence : DINT;
   C1_RemoteBrakeAndHomeSequenceAlarms : DINT;
   C1_RemoteBrakeAndHomeSequenceAlarmTimer : TIMER[32] := ([0].PRE := 300000, [1].PRE := 300000, [2].PRE := 300000, [3].PRE := 300000, [4].PRE := 300000, [5].PRE := 300000, [6].PRE := 300000, [7].PRE := 300000, [8].PRE := 300000, [9].PRE := 300000, [10].PRE := 300000);
   C1_RemoteBrakeAndHomeSequenceONS : BOOL;
   C1_RemoteBrakeTestCMD : BOOL;
   C1_RemoteDumpTestCMD : BOOL;
   C1_RemoteHomeCMD : BOOL;
   C1_RemoteScreenMessageNumber : DINT;
   C1_RemoteSequenceDelay : TIMER[8] := ([0].PRE := 2000, [1].PRE := 2000, [2].PRE := 2000, [3].PRE := 2000);
   C1_RevolutionCounter : COUNTER := (PRE := 60, ACC := 12);
   C1_ServoActionStatusOffDelay : TIMER := (PRE := 500, ACC := 500, EN := 1, DN := 1);
   C1_ServoActionStatusOnDelay : TIMER := (PRE := 500);
   C1_ServoFanOverload : ALIAS FOR C1_RIO_AENT:I.Data[1].2;
   C1_ServoStatus : BOOL;
   C1_SetEncoderHomePosition : BOOL;
   C1_SS_LocalRemote_1_IsRemote : ALIAS FOR C1_RIO_AENT:1:I.3;
   C1_SS_RemoteMode : BOOL := 1;
   C1_TargetPositionError : REAL := 7.247925e-05;
   C1_TargetPositionErrorTest : REAL := 7.247925e-05;
   C1_Warning : DINT := 67174464;
   C1DumpValveTestSequenceONS : DINT;
   C1HomeSensorTestMAM01 : MOTION_INSTRUCTION := (FLAGS := 704643072, DN := 1, PC := 1);
   C1HomeSequenceONS : BOOL;
   C1HomeSequenceONS2 : BOOL;
   C1ONS : DINT := 15;
   C2 : AXIS_SERVO_DRIVE;
   C2_32HourTimers : TIMER[4] := ([0].PRE := 115200000, [1].PRE := 115200000, [1].ACC := 1514379, [1].EN := 1, [1].TT := 1, [2].PRE := 115200000, [2].ACC := 11885390, [2].EN := 1, [2].TT := 1, [3].PRE := 115200000);
   C2_ActualPositionMOD60 : REAL := 41.785675;
   C2_All_DLY_OK : BOOL;
   C2_Brake_Daily_ok : BOOL;
   C2_Brake_Test_passed : BOOL;
   C2_BrakeReleaseSelected : BOOL;
   C2_BrakeSequenceInProcess : BOOL;
   C2_BrakeTest : BOOL;
   C2_BrakeTestEndPosition : REAL := 3.859576;
   C2_BrakeTestExpireTime : DINT := 32;
   C2_BrakeTestExpireTimeTemp : DINT := 115200000;
   C2_BrakeTestFailed : BOOL;
   C2_BrakeTestLocalDisable : BOOL;
   C2_BrakeTestMAJ01 : MOTION_INSTRUCTION := (FLAGS := 33554432);
   C2_BrakeTestMessageNumber : DINT;
   C2_BrakeTestONS : BOOL;
   C2_BrakeTestSelected : BOOL;
   C2_BrakeTestSequence : DINT;
   C2_BrakeTestSequenceAlarms : DINT;
   C2_BrakeTestSequenceAlarmTimer : TIMER[16] := ([1].PRE := 30000000, [2].PRE := 300000, [3].PRE := 300000, [4].PRE := 300000);
   C2_BrakeTestSequenceONS : DINT;
   C2_BrakeTestStartPosition : REAL := 1.1556641;
   C2_BrakeTestStoppingDistance : REAL := 2.7039118;
   C2_BrakeTestTimerHoldVel : TIMER := (PRE := 1000);
   C2_BrakeTestWarning : BOOL;
   C2_DisableTimer : TIMER := (PRE := 1000);
   C2_DistanceToEvac : REAL := 35.13733;
   C2_Dump_OK : BOOL;
   C2_DumpTest : BOOL;
   C2_DumpValveFailedOff : BOOL;
   C2_DumpValveFailedOn : BOOL;
   C2_DumpValveMessageNumber : DINT;
   C2_DumpValveReleaseSelected : BOOL;
   C2_DumpValveTestDelay : TIMER[4] := ([0].PRE := 20000, [1].PRE := 10000, [2].PRE := 5000, [3].PRE := 5000);
   C2_DumpValveTestDelay2 : TIMER := (PRE := 15000);
   C2_DumpValveTestExpireTime : DINT := 32;
   C2_DumpValveTestExpireTimeTemp : DINT := 115200000;
   C2_DumpValveTestSelected : BOOL;
   C2_DumpValveTestSequence : DINT;
   C2_DumpValveTestSequenceAlarms : DINT;
   C2_DumpValveTestSequenceAlarmTimer : TIMER[8] := ([0].PRE := 300000, [1].PRE := 300000);
   C2_EncoderCounts : DINT := 228023;
   C2_EncoderCountsRaw : ALIAS FOR C2_RIO_AENT:3:I.PresentData;
   C2_EncoderDegree : REAL := 341.72;
   C2_EncoderPositionAtHome : DINT := 4347022;
   C2_Error_Message_Raw : SINT[82] := ([0] := 64, [4] := 80, [5] := 104, [6] := 97, [7] := 115, [8] := 101, [9] := 32, [10] := 76, [11] := 111, [12] := 115, [13] := 115, [14] := 32, [15] := 70, [16] := 108, [17] := 116, [18] := 32, [19] := 32, [20] := 32);
   C2_EvacInPositionTest : DINT := 26810;
   C2_EvacPosition : REAL := 316.923;
   C2_EvacPositionMOD60 : REAL := 16.923004;
   C2_ExcecutePBHoldTimer : TIMER := (PRE := 5000);
   C2_FaultDebounce : TIMER[16] := ([0].PRE := 1250, [1].PRE := 500, [1].ACC := 500, [1].EN := 1, [1].DN := 1, [2].PRE := 1500, [3].PRE := 250, [4].PRE := 20);
   C2_FaultHoldTimer : TIMER[4] := ([0].PRE := 5000, [1].PRE := 5000);
   C2_FaultHomeSwitchNotFound : BOOL;
   C2_FaultStandard : DINT;
   C2_GoNearOnPathDelay : TIMER := (PRE := 2000);
   C2_GoToEvacMAM01 : MOTION_INSTRUCTION := (FLAGS := 33554432);
   C2_GoToOnPathMAM01 : MOTION_INSTRUCTION := (FLAGS := 704643072, DN := 1, PC := 1);
   C2_GoToOnPathMAM02 : MOTION_INSTRUCTION := (FLAGS := 33554432);
   C2_Home_OK : BOOL := 1;
   C2_Homed : BOOL := 1;
   C2_HomeDelay : TIMER[8] := ([0].PRE := 2000, [1].PRE := 2000, [2].PRE := 4000, [3].PRE := 2000, [4].PRE := 2000, [5].PRE := 1000, [6].PRE := 1000, [7].PRE := 3000);
   C2_HomeExpireTime : DINT := 31;
   C2_HomeExpireTimeTemp : DINT := 113686451;
   C2_HomeFindSwitchMAM01 : MOTION_INSTRUCTION := (FLAGS := 570425344, DN := 1);
   C2_HomeFindSwitchMAM02 : MOTION_INSTRUCTION := (FLAGS := 704643072, DN := 1, PC := 1);
   C2_HomeFindSwitchMAS01 : MOTION_INSTRUCTION := (FLAGS := 704643072, DN := 1, PC := 1);
   C2_HomeGetCloseToSwitchMAM01 : MOTION_INSTRUCTION := (FLAGS := 33554432);
   C2_HomeGoToOnPathMAM01 : MOTION_INSTRUCTION := (FLAGS := 704643072, DN := 1, PC := 1);
   C2_HomeInputStatus : BOOL := 1;
   C2_HomeMessageNumber : DINT := -2147483648;
   C2_HomeSensorTestMAM02 : MOTION_INSTRUCTION := (FLAGS := 704643072, DN := 1, PC := 1);
   C2_HomeSequence : DINT := -2147483648;
   C2_HomeSequenceAlarms : DINT;
   C2_HomeSequenceAlarmTimer : TIMER[32] := ([1].PRE := 300000, [2].PRE := 300000, [3].PRE := 300000, [4].PRE := 300000, [5].PRE := 300000, [6].PRE := 300000, [7].PRE := 300000, [8].PRE := 300000, [9].PRE := 300000, [10].PRE := 300000, [11].PRE := 300000, [12].PRE := 300000, [13].PRE := 300000, [14].PRE := 300000, [15].PRE := 300000, [16].PRE := 300000, [17].PRE := 300000, [18].PRE := 300000, [19].PRE := 300000, [20].PRE := 300000, [21].PRE := 300000, [22].PRE := 300000);
   C2_HomeSequenceInProcess : BOOL;
   C2_HomeSequenceMAH : MOTION_INSTRUCTION := (FLAGS := 671088640, DN := 1, PC := 1, STATE := 17);
   C2_HomeSwitchFaultK7KFailedOff : BOOL;
   C2_HomeSwitchFaultK7KFailedOn : BOOL;
   C2_HomeSwitchFaultSafeFailedOff : BOOL;
   C2_HomeSwitchFaultSafeFailedOn : BOOL;
   C2_HomeTest : REAL := 108.52835;
   C2_IndexEnable : BOOL;
   C2_IndexEnableTOF : TIMER := (PRE := 5000, ACC := 5001);
   C2_IndexMAM01 : MOTION_INSTRUCTION := (FLAGS := 33554432);
   C2_IndexMAS01 : MOTION_INSTRUCTION := (FLAGS := 33554432);
   C2_IndexMessageNumber : DINT;
   C2_IndexPermissive : BOOL;
   C2_Jog_ONS : DINT;
   C2_JogDirection : DINT;
   C2_JogEnable : BOOL;
   C2_JogEnableTOF : TIMER := (PRE := 15000, ACC := 15000);
   C2_JogForwardFastSelected : BOOL;
   C2_JogForwardSlowSelected : BOOL;
   C2_JogMAJ01 : MOTION_INSTRUCTION := (FLAGS := 570425344, DN := 1);
   C2_JogMAJ02 : MOTION_INSTRUCTION := (FLAGS := 33554432);
   C2_JogMAS01 : MOTION_INSTRUCTION := (FLAGS := 704643072, DN := 1, PC := 1);
   C2_JogMessageNumber : DINT;
   C2_JogPermissive : BOOL;
   C2_JogReverseFastSelected : BOOL;
   C2_JogReverseSlowSelected : BOOL;
   C2_LIM_ALARM_B : ALIAS FOR C2_RIO_AENT:I.Data[1].0;
   C2_LubricationMessageNumber : DINT;
   C2_LubricationOnTimer : TIMER := (PRE := 5000);
   C2_LubricationOverrideSelected : BOOL;
   C2_MAFR : MOTION_INSTRUCTION := (FLAGS := 301989888, ER := 1, ERR := 11);
   C2_MaintEnable : BOOL;
   C2_MAJAcceleration : REAL := 3.0;
   C2_MAJDeceleration : REAL := 5.0;
   C2_MAJSpeed : REAL := 8.5714;
   C2_MASR : MOTION_INSTRUCTION := (FLAGS := 33554432);
   C2_MotorActualPositionX1000 : DINT := 341786;
   C2_MotorAverageVelocityX1000 : DINT;
   C2_MotorFan : ALIAS FOR C2_RIO_AENT:O.Data[2].0;
   C2_MSF : MOTION_INSTRUCTION := (FLAGS := 536870912, DN := 1, STATUS := 2, STATE := 1);
   C2_MSO : MOTION_INSTRUCTION := (FLAGS := 536870912, DN := 1, STATE := 1);
   C2_Oiler : ALIAS FOR C2_RIO_AENT:O.Data[2].1;
   C2_OIT_BrakeRelease : BOOL;
   C2_OIT_BrakeReleaseDisplay : BOOL;
   C2_OIT_BrakeTest : BOOL;
   C2_OIT_BrakeTestDisplay : BOOL;
   C2_OIT_Command : DINT := 20;
   C2_OIT_Current : DINT := 20;
   C2_OIT_DumpValveRelease : BOOL;
   C2_OIT_DumpValveReleaseDisplay : BOOL;
   C2_OIT_DumpValveTest : BOOL;
   C2_OIT_DumpValveTestDisplay : BOOL;
   C2_OIT_FaultReset : BOOL;
   C2_OIT_FaultsExist : BOOL;
   C2_OIT_HomeCountDown : DINT := 6;
   C2_OIT_JogForwardFast : BOOL;
   C2_OIT_JogForwardFastDisplay : BOOL;
   C2_OIT_JogForwardSlow : BOOL;
   C2_OIT_JogForwardSlowDisplay : BOOL;
   C2_OIT_JogReverseFast : BOOL;
   C2_OIT_JogReverseFastDisplay : BOOL;
   C2_OIT_JogReverseSlow : BOOL;
   C2_OIT_JogReverseSlowDisplay : BOOL;
   C2_OIT_JogStopDisplay : BOOL := 1;
   C2_OIT_LubricationOverride : BOOL;
   C2_OIT_LubricationOverrideDisplay : BOOL;
   C2_OIT_PathError : DINT := -1992;
   C2_OIT_PathIndicatorHigh : DINT := 546;
   C2_OIT_PathIndicatorLow : DINT := -546;
   C2_OIT_WarningsExist : BOOL := 1;
   C2_OneTryToFixErrorONS : BOOL;
   C2_ONS : DINT;
   C2_ONS_Fault : DINT;
   C2_RemoteBrakeAndHomeSequence : DINT;
   C2_RemoteBrakeAndHomeSequenceAlarms : DINT;
   C2_RemoteBrakeAndHomeSequenceAlarmTimer : TIMER[8] := ([0].PRE := 300000, [1].PRE := 300000, [2].PRE := 300000, [3].PRE := 300000, [4].PRE := 300000, [5].PRE := 300000, [6].PRE := 300000);
   C2_RemoteBrakeAndHomeSequenceONS : BOOL;
   C2_RemoteBrakeTestCMD : BOOL;
   C2_RemoteDumpTestCMD : BOOL;
   C2_RemoteHomeCMD : BOOL;
   C2_RemoteScreenMessageNumber : DINT;
   C2_RemoteSequenceDelay : TIMER[4] := ([0].PRE := 2000, [1].PRE := 2000, [2].PRE := 2000);
   C2_RevolutionCounter : COUNTER := (PRE := 60, ACC := 45);
   C2_ServoActionStatusOffDelay : TIMER := (PRE := 500, ACC := 500, EN := 1, DN := 1);
   C2_ServoActionStatusOnDelay : TIMER := (PRE := 500);
   C2_ServoFanOverload : ALIAS FOR C2_RIO_AENT:I.Data[1].2;
   C2_ServoStatus : BOOL;
   C2_SetEncoderHomePosition : BOOL;
   C2_SS_LocalRemote_1_IsRemote : ALIAS FOR C2_RIO_AENT:I.Data[1].3;
   C2_SS_RemoteMode : BOOL := 1;
   C2_TargetPositionError : REAL := 4.196167e-05;
   C2_TargetPositionErrorTest : REAL := 4.196167e-05;
   C2_Warning : DINT := 67174464;
   C2DumpValveTestSequenceONS : DINT;
   C2HomeSensorTestMAM01 : MOTION_INSTRUCTION := (FLAGS := 704643072, DN := 1, PC := 1);
   C2HomeSequenceONS : BOOL;
   C2HomeSequenceONS2 : BOOL;
   C3 : AXIS_SERVO_DRIVE;
   C3_32HourTimers : TIMER[4] := ([0].PRE := 115200000, [1].PRE := 115200000, [1].ACC := 595930, [1].EN := 1, [1].TT := 1, [2].PRE := 115200000, [2].ACC := 11937189, [2].EN := 1, [2].TT := 1, [3].PRE := 115200000);
   C3_ActualPositionMOD60 : REAL := 41.785767;
   C3_All_DLY_OK : BOOL;
   C3_Brake_Daily_ok : BOOL;
   C3_Brake_Test_passed : BOOL := 1;
   C3_BrakeReleaseSelected : BOOL;
   C3_BrakeSequenceInProcess : BOOL;
   C3_BrakeTest : BOOL;
   C3_BrakeTestEndPosition : REAL := 6.837356;
   C3_BrakeTestExpireTime : DINT := 32;
   C3_BrakeTestExpireTimeTemp : DINT := 115200000;
   C3_BrakeTestFailed : BOOL;
   C3_BrakeTestLocalDisable : BOOL;
   C3_BrakeTestMAJ01 : MOTION_INSTRUCTION := (FLAGS := 33554432);
   C3_BrakeTestMessageNumber : DINT;
   C3_BrakeTestONS : BOOL;
   C3_BrakeTestSelected : BOOL;
   C3_BrakeTestSequence : DINT;
   C3_BrakeTestSequenceAlarms : DINT;
   C3_BrakeTestSequenceAlarmTimer : TIMER[16] := ([1].PRE := 30000000, [2].PRE := 300000, [3].PRE := 300000, [4].PRE := 300000);
   C3_BrakeTestSequenceONS : DINT;
   C3_BrakeTestStartPosition : REAL := 4.990414;
   C3_BrakeTestStoppingDistance : REAL := 1.846942;
   C3_BrakeTestTimerHoldVel : TIMER := (PRE := 1000);
   C3_BrakeTestWarning : BOOL;
   C3_DisableTimer : TIMER := (PRE := 1000);
   C3_DistanceToEvac : REAL := 37.473236;
   C3_Dump_OK : BOOL;
   C3_DumpTest : BOOL;
   C3_DumpValveFailedOff : BOOL;
   C3_DumpValveFailedOn : BOOL;
   C3_DumpValveMessageNumber : DINT;
   C3_DumpValveReleaseSelected : BOOL;
   C3_DumpValveTestDelay : TIMER[8] := ([0].PRE := 20000, [1].PRE := 10000, [2].PRE := 5000, [3].PRE := 5000);
   C3_DumpValveTestDelay2 : TIMER := (PRE := 15000);
   C3_DumpValveTestExpireTime : DINT := 32;
   C3_DumpValveTestExpireTimeTemp : DINT := 115200000;
   C3_DumpValveTestSelected : BOOL;
   C3_DumpValveTestSequence : DINT;
   C3_DumpValveTestSequenceAlarms : DINT;
   C3_DumpValveTestSequenceAlarmTimer : TIMER[16] := ([0].PRE := 300000, [1].PRE := 300000);
   C3_EncoderCounts : DINT := 524623;
   C3_EncoderCountsRaw : ALIAS FOR C3_RIO_AENT:3:I.PresentData;
   C3_EncoderDegree : REAL := 341.742;
   C3_EncoderPositionAtHome : DINT := 4367393;
   C3_Error_Message_Raw : SINT[82] := ([0] := 64, [4] := 80, [5] := 104, [6] := 97, [7] := 115, [8] := 101, [9] := 32, [10] := 76, [11] := 111, [12] := 115, [13] := 115, [14] := 32, [15] := 70, [16] := 108, [17] := 116, [18] := 32, [19] := 32, [20] := 32);
   C3_EvacInPositionTest : DINT := 19259;
   C3_EvacPosition : REAL := 19.259;
   C3_EvacPositionMOD60 : REAL := 19.259;
   C3_ExcecutePBHoldTimer : TIMER := (PRE := 5000);
   C3_FaultDebounce : TIMER[8] := ([0].PRE := 1250, [1].PRE := 500, [1].ACC := 500, [1].EN := 1, [1].DN := 1, [2].PRE := 1500, [3].PRE := 250, [4].PRE := 20);
   C3_FaultHoldTimer : TIMER[4] := ([0].PRE := 5000, [1].PRE := 5000);
   C3_FaultHomeSwitchNotFound : BOOL;
   C3_FaultStandard : DINT;
   C3_GoNearOnPathDelay : TIMER := (PRE := 2000);
   C3_GoToEvacMAM01 : MOTION_INSTRUCTION := (FLAGS := 33554432);
   C3_GoToOnPathMAM01 : MOTION_INSTRUCTION := (FLAGS := 704643072, DN := 1, PC := 1);
   C3_GoToOnPathMAM02 : MOTION_INSTRUCTION := (FLAGS := 33554432);
   C3_Home_OK : BOOL := 1;
   C3_Homed : BOOL := 1;
   C3_HomeDelay : TIMER[8] := ([0].PRE := 2000, [1].PRE := 2000, [2].PRE := 4000, [3].PRE := 2000, [4].PRE := 2000, [5].PRE := 1000, [6].PRE := 1000, [7].PRE := 3000);
   C3_HomeExpireTime : DINT := 31;
   C3_HomeExpireTimeTemp : DINT := 114604550;
   C3_HomeFindSwitchMAM01 : MOTION_INSTRUCTION := (FLAGS := 570425344, DN := 1);
   C3_HomeFindSwitchMAM02 : MOTION_INSTRUCTION := (FLAGS := 704643072, DN := 1, PC := 1);
   C3_HomeFindSwitchMAS01 : MOTION_INSTRUCTION := (FLAGS := 704643072, DN := 1, PC := 1);
   C3_HomeGetCloseToSwitchMAM01 : MOTION_INSTRUCTION := (FLAGS := 33554432);
   C3_HomeGoToOnPathMAM01 : MOTION_INSTRUCTION := (FLAGS := 704643072, DN := 1, PC := 1);
   C3_HomeInputStatus : BOOL := 1;
   C3_HomeMessageNumber : DINT := -2147483648;
   C3_HomeSensorTestMAM02 : MOTION_INSTRUCTION := (FLAGS := 704643072, DN := 1, PC := 1);
   C3_HomeSequence : DINT := -2147483648;
   C3_HomeSequenceAlarms : DINT;
   C3_HomeSequenceAlarmTimer : TIMER[32] := ([1].PRE := 300000, [2].PRE := 300000, [3].PRE := 300000, [4].PRE := 300000, [5].PRE := 300000, [6].PRE := 300000, [7].PRE := 300000, [8].PRE := 300000, [9].PRE := 300000, [10].PRE := 300000, [11].PRE := 300000, [12].PRE := 300000, [13].PRE := 300000, [14].PRE := 300000, [15].PRE := 300000, [16].PRE := 300000, [17].PRE := 300000, [18].PRE := 300000, [19].PRE := 300000, [20].PRE := 300000, [21].PRE := 300000, [22].PRE := 300000);
   C3_HomeSequenceInProcess : BOOL;
   C3_HomeSequenceMAH : MOTION_INSTRUCTION := (FLAGS := 671088640, DN := 1, PC := 1, STATE := 17);
   C3_HomeSwitchFaultK7KFailedOff : BOOL;
   C3_HomeSwitchFaultK7KFailedOn : BOOL;
   C3_HomeSwitchFaultSafeFailedOff : BOOL;
   C3_HomeSwitchFaultSafeFailedOn : BOOL;
   C3_HomeTest : REAL := -81.00246;
   C3_IndexEnable : BOOL;
   C3_IndexEnableTOF : TIMER := (PRE := 5000, ACC := 5000);
   C3_IndexMAM01 : MOTION_INSTRUCTION := (FLAGS := 33554432);
   C3_IndexMAS01 : MOTION_INSTRUCTION := (FLAGS := 33554432);
   C3_IndexMessageNumber : DINT;
   C3_IndexPermissive : BOOL;
   C3_Jog_ONS : DINT;
   C3_JogDirection : DINT;
   C3_JogEnable : BOOL;
   C3_JogEnableTOF : TIMER := (PRE := 15000, ACC := 15010);
   C3_JogForwardFastSelected : BOOL;
   C3_JogForwardSlowSelected : BOOL;
   C3_JogMAJ01 : MOTION_INSTRUCTION := (FLAGS := 570425344, DN := 1);
   C3_JogMAJ02 : MOTION_INSTRUCTION := (FLAGS := 33554432);
   C3_JogMAS01 : MOTION_INSTRUCTION := (FLAGS := 704643072, DN := 1, PC := 1);
   C3_JogMessageNumber : DINT;
   C3_JogPermissive : BOOL;
   C3_JogReverseFastSelected : BOOL;
   C3_JogReverseSlowSelected : BOOL;
   C3_LIM_ALARM_B : ALIAS FOR C3_RIO_AENT:I.Data[1].0;
   C3_LubricationMessageNumber : DINT;
   C3_LubricationOnTimer : TIMER := (PRE := 5000);
   C3_LubricationOverrideSelected : BOOL;
   C3_MAFR : MOTION_INSTRUCTION := (FLAGS := 536870912, DN := 1);
   C3_MAG : MOTION_INSTRUCTION := (FLAGS := 33554432);
   C3_MaintEnable : BOOL;
   C3_MAJAcceleration : REAL := 3.0;
   C3_MAJDeceleration : REAL := 5.0;
   C3_MAJSpeed : REAL := 8.5714;
   C3_MAS : MOTION_INSTRUCTION := (FLAGS := 33554432);
   C3_MASR : MOTION_INSTRUCTION := (FLAGS := 536870912, DN := 1);
   C3_MotorActualPositionX1000 : DINT := 341786;
   C3_MotorAverageVelocityX1000 : DINT;
   C3_MotorFan : ALIAS FOR C3_RIO_AENT:O.Data[2].0;
   C3_MSF : MOTION_INSTRUCTION := (FLAGS := 536870912, DN := 1, STATUS := 2, STATE := 1);
   C3_MSO : MOTION_INSTRUCTION := (FLAGS := 536870912, DN := 1, STATE := 1);
   C3_Oiler : ALIAS FOR C3_RIO_AENT:O.Data[2].1;
   C3_OIT_BrakeRelease : BOOL;
   C3_OIT_BrakeReleaseDisplay : BOOL;
   C3_OIT_BrakeTest : BOOL;
   C3_OIT_BrakeTestDisplay : BOOL;
   C3_OIT_Command : DINT := 20;
   C3_OIT_Current : DINT := 20;
   C3_OIT_DumpValveRelease : BOOL;
   C3_OIT_DumpValveReleaseDisplay : BOOL;
   C3_OIT_DumpValveTest : BOOL;
   C3_OIT_DumpValveTestDisplay : BOOL;
   C3_OIT_FaultReset : BOOL;
   C3_OIT_FaultsExist : BOOL;
   C3_OIT_HomeCountDown : DINT := 6;
   C3_OIT_JogForwardFast : BOOL;
   C3_OIT_JogForwardFastDisplay : BOOL;
   C3_OIT_JogForwardSlow : BOOL;
   C3_OIT_JogForwardSlowDisplay : BOOL;
   C3_OIT_JogReverseFast : BOOL;
   C3_OIT_JogReverseFastDisplay : BOOL;
   C3_OIT_JogReverseSlow : BOOL;
   C3_OIT_JogReverseSlowDisplay : BOOL;
   C3_OIT_JogStopDisplay : BOOL := 1;
   C3_OIT_LubricationOverride : BOOL;
   C3_OIT_LubricationOverrideDisplay : BOOL;
   C3_OIT_PathError : DINT := -2034;
   C3_OIT_PathIndicatorHigh : DINT := 546;
   C3_OIT_PathIndicatorLow : DINT := -546;
   C3_OIT_WarningsExist : BOOL := 1;
   C3_OneTryToFixErrorONS : BOOL;
   C3_ONS : DINT;
   C3_ONS_Fault : DINT;
   C3_RemoteBrakeAndHomeSequence : DINT;
   C3_RemoteBrakeAndHomeSequenceAlarms : DINT;
   C3_RemoteBrakeAndHomeSequenceAlarmTimer : TIMER[8] := ([0].PRE := 300000, [1].PRE := 300000, [2].PRE := 300000, [3].PRE := 300000, [4].PRE := 300000, [5].PRE := 300000, [6].PRE := 300000);
   C3_RemoteBrakeAndHomeSequenceONS : BOOL;
   C3_RemoteBrakeTestCMD : BOOL;
   C3_RemoteDumpTestCMD : BOOL;
   C3_RemoteHomeCMD : BOOL;
   C3_RemoteScreenMessageNumber : DINT;
   C3_RemoteSequenceDelay : TIMER[4] := ([0].PRE := 2000, [1].PRE := 2000, [2].PRE := 2000);
   C3_RevolutionCounter : COUNTER := (PRE := 60, ACC := 58);
   C3_ServoActionStatusOffDelay : TIMER := (PRE := 500, ACC := 510, EN := 1, DN := 1);
   C3_ServoActionStatusOnDelay : TIMER := (PRE := 500);
   C3_ServoFanOverload : ALIAS FOR C3_RIO_AENT:I.Data[1].2;
   C3_ServoStatus : BOOL;
   C3_SetEncoderHomePosition : BOOL;
   C3_SS_LocalRemote_1_IsRemote : ALIAS FOR C3_RIO_AENT:1:I.3;
   C3_SS_RemoteMode : BOOL := 1;
   C3_TargetPositionError : REAL := -4.9591064e-05;
   C3_TargetPositionErrorTest : REAL := -4.9591064e-05;
   C3_Warning : DINT := 67174464;
   C3DumpValveTestSequenceONS : DINT;
   C3HomeSensorTestMAM01 : MOTION_INSTRUCTION := (FLAGS := 704643072, DN := 1, PC := 1);
   C3HomeSequenceONS : BOOL;
   C3HomeSequenceONS2 : BOOL;
   Carsl2_Fault_Reset : BOOL;
   Carsl3_Fault_Reset : BOOL;
   DeviceNet_OK : BOOL := 1;
   ErrorMinMaxTotal : REAL[4];
   GroupResetONS : DINT;
   GSV_BSL : CONTROL := (LEN := 1);
   GSV_BSL_Array : DINT[2] := ([0] := 536870912);
   GSVTimer : TIMER := (PRE := 100, ACC := 40, EN := 1, TT := 1);
   JoeEnableSERCOScOut : BOOL;
   MasterAtSpeed : BOOL;
   MasterClockCopyMAJ : MOTION_INSTRUCTION := (FLAGS := 33554432);
   MasterClockCopyMAS_Stop1 : MOTION_INSTRUCTION := (FLAGS := 33554432);
   MasterClockCopyMAS_Stop2 : MOTION_INSTRUCTION := (FLAGS := 33554432);
   MasterClockCopyMRP : MOTION_INSTRUCTION := (FLAGS := 570425344, DN := 1);
   MasterClockLocal : AXIS_VIRTUAL;
   MasterClockLocalActualPosition : DINT := 39875;
   MasterClockLocalCorrectionAmount : REAL;
   MasterClockTagetTicks : REAL := 4875.0;
   MasterCorrectionStartDelay : TIMER := (PRE := 5000);
   MasterError : REAL;
   MasterErrorCorrectionAtStartONS : BOOL;
   MasterErrorMaxCheck : REAL;
   MasterErrorMinCheck : REAL;
   MasterMinMaxCheck : TIMER := (PRE := 15000);
   MESSAGE_SERCOScOut : MESSAGE;
        MessageParameters(ServiceCode := 16#0051, LocalElement := servicecode[0], DestinationTag := respcode[0], ...)
   Motion : MOTION_GROUP;
   MotionMSGR : MOTION_INSTRUCTION := (FLAGS := 570425344, DN := 1);
   MS_ENBT : DINT[10] := ([0] := 16384, [1] := 16384, [2] := 16384, [3] := 16384, [4] := 16384, [5] := 16384, [6] := 16384, [7] := 16384);
   MS_ENBTRaw : DINT[10] := ([0] := 16#0000_4201, [1] := 16#0000_4201, [2] := 16#0000_4201, [3] := 16#0000_4201, [4] := 16#0000_4201, [5] := 16#0000_4201, [6] := 16#0000_4201, [7] := 16#0000_4202);
   Multiplier : DINT := 26;
   none : BOOL;
   NoScan_Comment : BOOL;
   Ons_Fault : DINT;
   ONS_STFault : DINT;
   ProcFaultWord : DINT;
   ProcForceEn : ALIAS FOR ProcForceStatus.1;
   ProcForceExist : ALIAS FOR ProcForceStatus.0;
   ProcForceStatus : DINT;
   ProcLoBattery : ALIAS FOR ProcFaultWord.10;
   ProcRem : BOOL := 1;
   ProcRun : BOOL;
   ProcStatus : DINT := 12384;
   Rail_Bypass1 : ALIAS FOR SSC01_Safe1:I.Pt06Data;
   Rail_Bypass2 : ALIAS FOR SSC01_Safe1:I.Pt07Data;
   Rail_Bypass_RIN : REDUNDANT_INPUT := (ChannelA := 1, ChannelB := 1, O1 := 1);
   RAIL_ENABLE_LH1 : ALIAS FOR SSC01_Safe1:I.Pt00Data;
   RAIL_ENABLE_LH2 : ALIAS FOR SSC01_Safe1:I.Pt01Data;
   RAIL_ENABLE_LH3 : ALIAS FOR SSC01_Safe1:I.Pt02Data;
   RAIL_ENABLE_RH1 : ALIAS FOR SSC01_Safe1:I.Pt03Data;
   RAIL_ENABLE_RH2 : ALIAS FOR SSC01_Safe1:I.Pt04Data;
   RAIL_ENABLE_RH3 : ALIAS FOR SSC01_Safe1:I.Pt05Data;
   RAIL_SHUNT_FDBK_LH1 : ALIAS FOR SSC01_Safe3:I.Pt00Data;
   RAIL_SHUNT_FDBK_LH2 : ALIAS FOR SSC01_Safe3:I.Pt01Data;
   RAIL_SHUNT_FDBK_LH3 : ALIAS FOR SSC01_Safe3:I.Pt02Data;
   Rail_Shunt_Fdbk_OK : BOOL := 1;
   RAIL_SHUNT_FDBK_RH1 : ALIAS FOR SSC01_Safe3:I.Pt03Data;
   RAIL_SHUNT_FDBK_RH2 : ALIAS FOR SSC01_Safe3:I.Pt04Data;
   RAIL_SHUNT_FDBK_RH3 : ALIAS FOR SSC01_Safe3:I.Pt05Data;
   RAIL_SHUNT_LH1 : ALIAS FOR SSC01_Safe1:O.Pt00Data;
   RAIL_SHUNT_LH2 : ALIAS FOR SSC01_Safe1:O.Pt01Data;
   RAIL_SHUNT_LH3 : ALIAS FOR SSC01_Safe1:O.Pt02Data;
   RAIL_SHUNT_RH1 : ALIAS FOR SSC01_Safe1:O.Pt03Data;
   RAIL_SHUNT_RH2 : ALIAS FOR SSC01_Safe1:O.Pt04Data;
   RAIL_SHUNT_RH3 : ALIAS FOR SSC01_Safe1:O.Pt05Data;
   RCS_CMD_Auto_TON : TIMER := (PRE := 5950);
   RCS_CMD_BrakeTest : BOOL;
   RCS_CMD_BrakeTest_TON : TIMER := (PRE := 1000);
   RCS_CMD_Evac_TON : TIMER := (PRE := 5900);
   RCS_CMD_EvacToStation : BOOL;
   RCS_CMD_GoNearOnPath : BOOL;
   RCS_CMD_GoNearOnPath_TON : TIMER := (PRE := 1000);
   RCS_Cmd_Mismatch_TON : TIMER := (PRE := 500);
   RCS_CMD_RunInAuto : BOOL;
   RCS_CMD_Stop1 : BOOL := 1;
   RCS_CMD_Stop2 : BOOL;
   RCS_CMD_Stop_TON : TIMER := (PRE := 1500, ACC := 1500, EN := 1, DN := 1);
   RCS_Cmd_Unknown : BOOL;
   RCS_MasterClock : ALIAS FOR RCS_SafeMemory_S01.Master_Clock;
   RCS_MasterClockLocalTagetDegrees : REAL := 41.785717;
   RCS_MasterPositionMOD7000 : DINT := 1336;
   RCS_MasterPositionMOD7000X1000 : DINT := 1336000;
   RCS_MotionEnable_TON : TIMER := (PRE := 25);
   RCS_OnPathEnable_TON : TIMER := (PRE := 2000);
   RCS_PwrDisc_AuxA : BOOL := 1;
   RCS_PwrDisc_AuxB : BOOL := 1;
   RCS_PwrDisc_RIN : REDUNDANT_INPUT := (ChannelA := 1, ChannelB := 1, O1 := 1);
   RCS_PwrDiscA : ALIAS FOR SSC01_Safe2:I.Pt04Data;
   RCS_PwrDiscB : ALIAS FOR SSC01_Safe2:I.Pt05Data;
   RCS_SafeMemory_S01 : Udt_RCS_SafeData := (Status.ConnectionFaulted := 1, RailStateEthernet := 2);
   RCS_SyncMotionEnable : BOOL;
   RCSMasterGearMAM02 : MOTION_INSTRUCTION := (FLAGS := 33554432);
   respcode : INT[1];
   S1_C1_SafeOffFdbkRIN : REDUNDANT_INPUT := (ChannelA := 1, ChannelB := 1, O1 := 1);
   S1_C3_SafeOffFdbkRIN : REDUNDANT_INPUT := (ChannelA := 1, ChannelB := 1, O1 := 1);
   S_C01_MStopOK : BOOL;
   S_C02_MStopOK : BOOL;
   S_C03_MStopOK : BOOL;
   S_C1_AtEvacSpeed : BOOL;
   S_C1_BrakeRelease : ALIAS FOR C1_Safe:O.Pt06Data;
   S_C1_BrakeReleaseSelected : BOOL;
   S_C1_BrakeTest : BOOL;
   S_C1_CircuitReset : BOOL;
   S_C1_CircuitReset_Pulse : TIMER := (PRE := 25, ACC := 27);
   S_C1_DrawBridge_LS1 : ALIAS FOR SSC01_Safe2:I.Pt00Data;
   S_C1_DrawBridge_LS2 : ALIAS FOR SSC01_Safe2:I.Pt01Data;
   S_C1_DrawbridgeInputOK : BOOL := 1;
   S_C1_DrawbridgeRIN : REDUNDANT_INPUT := (ChannelA := 1, ChannelB := 1, O1 := 1);
   S_C1_DumpTest : BOOL;
   S_C1_DumpValveRelease : ALIAS FOR C1_Safe:O.Pt05Data;
   S_C1_DumpValveReleaseSelected : BOOL;
   S_C1_EncoderBuffer : DINT[4] := ([0] := 481762, [1] := 481762);
   S_C1_EncoderChange : DINT;
   S_C1_EncoderCounter : DINT := 4720180;
   S_C1_EncoderCounts : DINT := 481762;
   S_C1_EncoderPositionAtHome : DINT := 4345814;
   S_C1_EncoderPositionAtHomeSet : BOOL;
   S_C1_EncoderPositionDegree : DINT := 289639;
   S_C1_EncoderRev : DINT := 321709;
   S_C1_EncoderRevX1000 : DINT := 321709000;
   S_C1_EncoderTemp : DINT;
   S_C1_EncoderTemp2 : DINT;
   S_C1_EvacOk : BOOL := 1;
   S_C1_ExecuteInputOK : BOOL := 1;
   S_C1_ExecutePB : BOOL;
   S_C1_FaultReset : BOOL;
   S_C1_FaultSafety : DINT;
   S_C1_FaultSafety_OK : BOOL := 1;
   S_C1_FaultStandard : DINT;
   S_C1_FaultStandard_OK : BOOL := 1;
   S_C1_FaultTimer : TIMER[8] := ([0].PRE := 100, [1].PRE := 1500, [2].PRE := 1500, [3].PRE := 200);
   S_C1_FW_LocalOK : BOOL := 1;
   S_C1_Homed : BOOL;
   S_C1_HomeInputStatus : BOOL := 1;
   S_C1_HomeSafePE : ALIAS FOR C1_Safe:I.Pt04Data;
   S_C1_HomeSequenceInProcess : BOOL;
   S_C1_InEvacPosition : BOOL := 1;
   S_C1_MaintEnable : BOOL;
   S_C1_MCC1_LIM_MCR : ALIAS FOR C1_Safe:O.Pt04Data;
   S_C1_ModeLocal : BOOL;
   S_C1_ModeRemote : BOOL := 1;
   S_C1_MotionEnabled : BOOL;
   S_C1_MOTN_EXEC_RIN : REDUNDANT_INPUT;
   S_C1_MOTN_EXEC_SS_A : ALIAS FOR C1_Safe:I.Pt02Data;
   S_C1_MOTN_EXEC_SS_B : ALIAS FOR C1_Safe:I.Pt03Data;
   S_C1_MotorActualPositionX1000 : DINT := 289785;
   S_C1_MotorActualPositionX1000MOD60 : DINT := 49785;
   S_C1_MotorAverageVelocityX1000 : DINT;
   S_C1_MotorToEncoderError : DINT := -146;
   S_C1_MStop : EMERGENCY_STOP := (ResetType := 1, ChannelA := 1, ChannelB := 1, O1 := 1);
   S_C1_MSTOP_A : ALIAS FOR C1_Safe:I.Pt06Data;
   S_C1_MSTOP_B : ALIAS FOR C1_Safe:I.Pt07Data;
   S_C1_MSTOP_InputOK : BOOL := 1;
   S_C1_MSTOP_LT : ALIAS FOR C1_Safe:O.Pt02Data;
   S_C1_NearOnPath : BOOL;
   S_C1_NearOnPathHi : DINT := 3500;
   S_C1_NearOnPathHiBase : DINT := 3500;
   S_C1_NearOnPathLow : DINT := -3500;
   S_C1_NearOnPathLowBase : DINT := -3500;
   S_C1_OffPath : BOOL := 1;
   S_C1_OIT_FaultReset : BOOL;
   S_C1_OnPath : BOOL;
   S_C1_OnPathHi : DINT := 214;
   S_C1_OnPathLow : DINT := -214;
   S_C1_ONS : DINT := 16;
   S_C1_ONS_CircuitFault : BOOL := 1;
   S_C1_ONS_Fault : BOOL;
   S_C1_ONS_Status : BOOL;
   S_C1_OutputEnable : BOOL;
   S_C1_PathError : DINT := 21666;
   S_C1_PathErrorTest : DINT := -38334;
   S_C1_PathErrorTestTemp : DINT := 10215;
   S_C1_PathErrorTestTemp2 : DINT := 11357;
   S_C1_PathOffset : DINT;
   S_C1_PressureOK : ALIAS FOR C1_Safe:I.Pt05Data;
   S_C1_RemoteBrakeAndHomeSequence : DINT;
   S_C1_ResetTOF : TIMER := (PRE := 500, ACC := 500);
   S_C1_ReverseMotionDebounce : TIMER := (PRE := 500);
   S_C1_SAFE_FDBK_Aux1 : BOOL := 1;
   S_C1_SAFE_FDBK_Aux2 : BOOL := 1;
   S_C1_SAFE_OFF_FDBK1 : ALIAS FOR C1_Safe:I.Pt01Data;
   S_C1_SAFE_OFF_FDBK2 : ALIAS FOR C1_Safe:I.Pt00Data;
   S_C1_SafeOff_ROUT : REDUNDANT_OUTPUT := (Feedback1 := 1, Feedback2 := 1);
   S_C1_SafeOffEnabled : BOOL;
   S_C1_SafeOffEngaged : BOOL := 1;
   S_C1_SafeOffInputOK : BOOL := 1;
   S_C1_SAFETY_ENABLE_1 : ALIAS FOR C1_Safe:O.Pt00Data;
   S_C1_SAFETY_ENABLE_2 : ALIAS FOR C1_Safe:O.Pt01Data;
   S_C1_ServoStatus : BOOL;
   S_C1_SetEncoderHomePosition : BOOL;
   S_C1_SS_RemoteMode : BOOL := 1;
   S_C1_Stop0 : BOOL;
   S_C1_Stop0_OK : BOOL := 1;
   S_C1_Stop1 : BOOL := 1;
   S_C1_Stop1_OK : BOOL := 1;
   S_C1_Stop1_OK_TOF : TIMER := (PRE := 1000, EN := 1, DN := 1);
   S_C1_WindowAdderTemp1 : DINT := 72;
   S_C1_WindowAdderTemp2 : DINT := 38059;
   S_C1_WindowAdderTemp3 : DINT := 38;
   S_C2_AtEvacSpeed : BOOL;
   S_C2_BrakeRelease : ALIAS FOR C2_Safe:O.Pt06Data;
   S_C2_BrakeReleaseSelected : BOOL;
   S_C2_BrakeTest : BOOL;
   S_C2_CircuitReset : BOOL;
   S_C2_CircuitReset_Pulse : TIMER := (ACC := 27);
   S_C2_DrawBridge_LS1 : ALIAS FOR SSC01_Safe2:I.Pt02Data;
   S_C2_DrawBridge_LS2 : ALIAS FOR SSC01_Safe2:I.Pt03Data;
   S_C2_DrawbridgeInputOK : BOOL := 1;
   S_C2_DrawbridgeRIN : REDUNDANT_INPUT := (ChannelA := 1, ChannelB := 1, O1 := 1);
   S_C2_DumpTest : BOOL;
   S_C2_DumpValveRelease : ALIAS FOR C2_Safe:O.Pt05Data;
   S_C2_DumpValveReleaseSelected : BOOL;
   S_C2_EncoderBuffer : DINT[4] := ([0] := 821317, [1] := 821317);
   S_C2_EncoderChange : DINT;
   S_C2_EncoderCounter : DINT := 4361529;
   S_C2_EncoderCounts : DINT := 821317;
   S_C2_EncoderPositionAtHome : DINT := 4347022;
   S_C2_EncoderPositionAtHomeSet : BOOL;
   S_C2_EncoderPositionDegree : DINT := 326741;
   S_C2_EncoderRev : DINT := 362919;
   S_C2_EncoderRevX1000 : DINT := 362919000;
   S_C2_EncoderTemp : DINT;
   S_C2_EncoderTemp2 : DINT;
   S_C2_EvacOK : BOOL;
   S_C2_ExecuteInputOK : BOOL := 1;
   S_C2_ExecutePB : BOOL;
   S_C2_FaultReset : BOOL;
   S_C2_FaultSafety : DINT := 1073741824;
   S_C2_FaultSafety_OK : BOOL;
   S_C2_FaultStandard : DINT;
   S_C2_FaultStandard_OK : BOOL := 1;
   S_C2_FaultTimer : TIMER[8] := ([0].PRE := 100, [1].PRE := 1500, [2].PRE := 1500, [3].PRE := 200);
   S_C2_FW_LocalOK : BOOL := 1;
   S_C2_Homed : BOOL := 1;
   S_C2_HomeInputStatus : BOOL := 1;
   S_C2_HomeSafePE : ALIAS FOR C2_Safe:I.Pt04Data;
   S_C2_HomeSequenceInProcess : BOOL;
   S_C2_InEvacPosition : BOOL;
   S_C2_MaintEnable : BOOL;
   S_C2_MCC2_LIM_MCR : ALIAS FOR C2_Safe:O.Pt04Data;
   S_C2_ModeLocal : BOOL;
   S_C2_ModeRemote : BOOL := 1;
   S_C2_MotionEnabled : BOOL;
   S_C2_MOTN_EXEC_RIN : REDUNDANT_INPUT;
   S_C2_MOTN_EXEC_SS_A : ALIAS FOR C2_Safe:I.Pt02Data;
   S_C2_MOTN_EXEC_SS_B : ALIAS FOR C2_Safe:I.Pt03Data;
   S_C2_MotorActualPositionX1000 : DINT := 326810;
   S_C2_MotorActualPositionX1000MOD60 : DINT := 26810;
   S_C2_MotorAverageVelocityX1000 : DINT;
   S_C2_MotorToEncoderError : DINT := -69;
   S_C2_MStop : EMERGENCY_STOP := (ResetType := 1, ChannelA := 1, ChannelB := 1, O1 := 1);
   S_C2_MSTOP_A : ALIAS FOR C2_Safe:I.Pt06Data;
   S_C2_MSTOP_B : ALIAS FOR C2_Safe:I.Pt07Data;
   S_C2_MSTOP_InputOK : BOOL := 1;
   S_C2_MSTOP_LT : ALIAS FOR C2_Safe:O.Pt02Data;
   S_C2_NearOnPath : BOOL;
   S_C2_NearOnPathHi : DINT := 3500;
   S_C2_NearOnPathHiBase : DINT := 3500;
   S_C2_NearOnPathLow : DINT := -3500;
   S_C2_NearOnPathLowBase : DINT := -3500;
   S_C2_OffPath : BOOL := 1;
   S_C2_OIT_FaultReset : BOOL;
   S_C2_OnPath : BOOL;
   S_C2_OnPathHi : DINT := 214;
   S_C2_OnPathLow : DINT := -214;
   S_C2_ONS : DINT := 16;
   S_C2_ONS_CircuitFault : BOOL := 1;
   S_C2_ONS_Fault : BOOL;
   S_C2_ONS_Status : BOOL;
   S_C2_OutputEnable : BOOL;
   S_C2_PathError : DINT := -15359;
   S_C2_PathErrorTest : DINT := -15359;
   S_C2_PathErrorTestTemp : DINT := 55;
   S_C2_PathErrorTestTemp2 : DINT := 206;
   S_C2_PathOffset : DINT;
   S_C2_PressureOK : ALIAS FOR C2_Safe:I.Pt05Data;
   S_C2_RemoteBrakeAndHomeSequence : DINT;
   S_C2_ResetTOF : TIMER := (PRE := 500, ACC := 500);
   S_C2_ReverseMotionDebounce : TIMER := (PRE := 500);
   S_C2_SAFE_FDBK_Aux1 : BOOL := 1;
   S_C2_SAFE_FDBK_Aux2 : BOOL := 1;
   S_C2_SAFE_OFF_FDBK1 : ALIAS FOR C2_Safe:I.Pt01Data;
   S_C2_SAFE_OFF_FDBK2 : ALIAS FOR C2_Safe:I.Pt00Data;
   S_C2_SafeOff_ROUT : REDUNDANT_OUTPUT := (Feedback1 := 1, Feedback2 := 1);
   S_C2_SafeOffEnabled : BOOL;
   S_C2_SafeOffEngaged : BOOL := 1;
   S_C2_SafeOffFdbkRIN : REDUNDANT_INPUT := (ChannelA := 1, ChannelB := 1, O1 := 1);
   S_C2_SafeOffInputOK : BOOL := 1;
   S_C2_SAFETY_ENABLE_1 : ALIAS FOR C2_Safe:O.Pt00Data;
   S_C2_SAFETY_ENABLE_2 : ALIAS FOR C2_Safe:O.Pt01Data;
   S_C2_ServoStatus : BOOL;
   S_C2_SetEncoderHomePosition : BOOL;
   S_C2_SS_RemoteMode : BOOL := 1;
   S_C2_Stop0 : BOOL := 1;
   S_C2_Stop0_OK : BOOL := 1;
   S_C2_Stop1 : BOOL;
   S_C2_Stop1_OK : BOOL;
   S_C2_Stop1_OK_TOF : TIMER := (PRE := 1000, ACC := 1000);
   S_C2_WindowAdderTemp1 : DINT := 5;
   S_C2_WindowAdderTemp2 : DINT := 2643;
   S_C2_WindowAdderTemp3 : DINT := 2;
   S_C3_AtEvacSpeed : BOOL;
   S_C3_BrakeRelease : ALIAS FOR C3_Safe:O.Pt06Data;
   S_C3_BrakeReleaseSelected : BOOL;
   S_C3_BrakeTest : BOOL;
   S_C3_CircuitReset : BOOL;
   S_C3_CircuitReset_Pulse : TIMER := (PRE := 25, ACC := 27);
   S_C3_DrawBridge_LS1 : ALIAS FOR SSC01_Safe2:I.Pt06Data;
   S_C3_DrawBridge_LS2 : ALIAS FOR SSC01_Safe2:I.Pt07Data;
   S_C3_DrawbridgeInputOK : BOOL := 1;
   S_C3_DrawbridgeRIN : REDUNDANT_INPUT := (ChannelA := 1, ChannelB := 1, O1 := 1);
   S_C3_DumpTest : BOOL;
   S_C3_DumpValveRelease : ALIAS FOR C3_Safe:O.Pt05Data;
   S_C3_DumpValveReleaseSelected : BOOL;
   S_C3_EncoderBuffer : DINT[4] := ([0] := 752371, [1] := 752371);
   S_C3_EncoderChange : DINT;
   S_C3_EncoderCounter : DINT := 4419803;
   S_C3_EncoderCounts : DINT := 752371;
   S_C3_EncoderDegree : DINT := 19205;
   S_C3_EncoderPositionAtHome : DINT := 4367393;
   S_C3_EncoderPositionAtHomeSet : BOOL;
   S_C3_EncoderRev : DINT := 21332;
   S_C3_EncoderRevX1000 : DINT := 21332000;
   S_C3_EncoderTemp : DINT;
   S_C3_EncoderTemp2 : DINT;
   S_C3_EvacOK : BOOL := 1;
   S_C3_ExecuteInputOK : BOOL := 1;
   S_C3_ExecutePB : BOOL;
   S_C3_FaultReset : BOOL;
   S_C3_FaultSafety : DINT;
   S_C3_FaultSafety_OK : BOOL := 1;
   S_C3_FaultStandard : DINT;
   S_C3_FaultStandard_OK : BOOL := 1;
   S_C3_FaultTimer : TIMER[8] := ([0].PRE := 100, [1].PRE := 1500, [2].PRE := 1500, [3].PRE := 200);
   S_C3_FW_LocalOK : BOOL := 1;
   S_C3_Homed : BOOL := 1;
   S_C3_HomeInputStatus : BOOL := 1;
   S_C3_HomeSafePE : ALIAS FOR C3_Safe:I.Pt04Data;
   S_C3_HomeSequenceInProcess : BOOL;
   S_C3_InEvacPosition : BOOL := 1;
   S_C3_MaintEnable : BOOL;
   S_C3_MCC3_LIM_MCR : ALIAS FOR C3_Safe:O.Pt04Data;
   S_C3_ModeLocal : BOOL;
   S_C3_ModeRemote : BOOL := 1;
   S_C3_MotionEnabled : BOOL;
   S_C3_MOTN_EXEC_RIN : REDUNDANT_INPUT;
   S_C3_MOTN_EXEC_SS_A : ALIAS FOR C3_Safe:I.Pt02Data;
   S_C3_MOTN_EXEC_SS_B : ALIAS FOR C3_Safe:I.Pt03Data;
   S_C3_MotorActualPositionX1000 : DINT := 19259;
   S_C3_MotorActualPositionX1000MOD60 : DINT := 19259;
   S_C3_MotorAverageVelocityX1000 : DINT;
   S_C3_MotorToEncoderError : DINT := -54;
   S_C3_MStop : EMERGENCY_STOP := (ResetType := 1, ChannelA := 1, ChannelB := 1, O1 := 1);
   S_C3_MSTOP_A : ALIAS FOR C3_Safe:I.Pt06Data;
   S_C3_MSTOP_B : ALIAS FOR C3_Safe:I.Pt07Data;
   S_C3_MSTOP_InputOK : BOOL := 1;
   S_C3_MSTOP_LT : ALIAS FOR C3_Safe:O.Pt02Data;
   S_C3_NearOnPath : BOOL;
   S_C3_NearOnPathHi : DINT := 3500;
   S_C3_NearOnPathHiBase : DINT := 3500;
   S_C3_NearOnPathLow : DINT := -3500;
   S_C3_NearOnPathLowBase : DINT := -3500;
   S_C3_OffPath : BOOL := 1;
   S_C3_OIT_FaultReset : BOOL;
   S_C3_OnPath : BOOL;
   S_C3_OnPathHi : DINT := 214;
   S_C3_OnPathLow : DINT := -214;
   S_C3_ONS : DINT := 16;
   S_C3_ONS_CircuitFault : BOOL := 1;
   S_C3_ONS_Fault : BOOL;
   S_C3_ONS_Status : BOOL;
   S_C3_OutputEnable : BOOL;
   S_C3_PathError : DINT := -7808;
   S_C3_PathErrorTest : DINT := -7808;
   S_C3_PathErrorTestTemp : DINT := 134;
   S_C3_PathErrorTestTemp2 : DINT := 206;
   S_C3_PathOffset : DINT;
   S_C3_PressureOK : ALIAS FOR C3_Safe:I.Pt05Data;
   S_C3_RemoteBrakeAndHomeSequence : DINT;
   S_C3_ResetTOF : TIMER := (PRE := 500, ACC := 500);
   S_C3_ReverseMotionDebounce : TIMER := (PRE := 500);
   S_C3_SAFE_FDBK_Aux1 : BOOL := 1;
   S_C3_SAFE_FDBK_Aux2 : BOOL := 1;
   S_C3_SAFE_OFF_FDBK1 : ALIAS FOR C3_Safe:I.Pt01Data;
   S_C3_SAFE_OFF_FDBK2 : ALIAS FOR C3_Safe:I.Pt00Data;
   S_C3_SafeOff_ROUT : REDUNDANT_OUTPUT := (Feedback1 := 1, Feedback2 := 1);
   S_C3_SafeOffEnabled : BOOL;
   S_C3_SafeOffEngaged : BOOL := 1;
   S_C3_SafeOffInputOK : BOOL := 1;
   S_C3_SAFETY_ENABLE_1 : ALIAS FOR C3_Safe:O.Pt00Data;
   S_C3_SAFETY_ENABLE_2 : ALIAS FOR C3_Safe:O.Pt01Data;
   S_C3_ServoStatus : BOOL;
   S_C3_SetEncoderHomePosition : BOOL;
   S_C3_SS_RemoteMode : BOOL := 1;
   S_C3_Stop0 : BOOL := 1;
   S_C3_Stop0_OK : BOOL := 1;
   S_C3_Stop1 : BOOL;
   S_C3_Stop1_OK : BOOL := 1;
   S_C3_Stop1_OK_TOF : TIMER := (PRE := 1000, EN := 1, DN := 1);
   S_C3_WindowAdderTemp1 : DINT := 31;
   S_C3_WindowAdderTemp2 : DINT := 16387;
   S_C3_WindowAdderTemp3 : DINT := 16;
   S_DeviceNet_OK : BOOL := 1;
   S_EncoderCtsFor360Deg : DINT := 399861;
   S_EncoderRollover : DINT := 1044480;
   S_EvacToStationTON : TIMER := (PRE := 9000);
   S_FaultReset : BOOL;
   S_FlashOff : TIMER := (PRE := 500, ACC := 227, EN := 1, TT := 1);
   S_FlashOn : TIMER := (PRE := 500, ACC := 500, EN := 1, DN := 1);
   S_MasterClockLocalActualPosition : DINT := 5675;
   S_ONS : BOOL := 1;
   S_RailStateHardware : DINT;
   S_RCS_CMD_FaultReset : BOOL;
   S_RCS_EvacSpeedStart_TON : TIMER := (PRE := 15000);
   S_RCS_MasterPositionDegrees : DINT := 11451;
   S_RCS_MotionCMD_Auto : BOOL;
   S_RCS_MotionCMD_BrakeTest : BOOL;
   S_RCS_MotionCMD_Evac : BOOL;
   S_RCS_MotionCMD_GoNearOnPath : BOOL;
   S_RCS_MotionCMD_Stop1 : BOOL := 1;
   S_RCS_MotionCMD_Stop2 : BOOL;
   S_RCS_MotionEnable : BOOL;
   S_RCS_RailStateEthernet : ALIAS FOR RCS_SafeMemory_S01.RailStateEthernet;
   S_RCS_RailStateHardwareUnknown : DINT := 62;
   S_S01_Mode_Remote : BOOL := 1;
   S_S01_NearOnPath : BOOL;
   S_S01_OnPath : BOOL;
   S_S01_Ready : BOOL;
   S_SSC_InputsOK : BOOL := 1;
   S_System_FaultStandard : DINT;
   SafetySignatureGSVTimer : TIMER := (PRE := 3600000, ACC := 3318090, EN := 1, TT := 1);
   SafetySignatureSINT : SINT[50] := ([0] := 37, [4] := 50, [5] := 65, [6] := 56, [7] := 54, [8] := 57, [9] := 54, [10] := 65, [11] := 51, [12] := 44, [13] := 32, [14] := 48, [15] := 53, [16] := 47, [17] := 49, [18] := 53, [19] := 47, [20] := 50, [21] := 48, [22] := 49, [23] := 48, [24] := 44, [25] := 32, [26] := 48, [27] := 48, [28] := 58, [29] := 51, [30] := 54, [31] := 58, [32] := 50, [33] := 50, [34] := 46, [35] := 55, [36] := 55, [37] := 48, [38] := 32, [39] := 65, [40] := 77);
   SafetySignatureString : STRING := '2A8696A3, 05/15/2010, 00:36:22.770 AM';
   servicecode : INT[1];
   SSC_Auto_Decel1 : BOOL;
   SSC_Mode_Local_LT : ALIAS FOR SSC01_Safe3:O.Pt00Data;
   SSC_Mode_Remote_LT : ALIAS FOR SSC01_Safe3:O.Pt02Data;
   SSC_NoStopFault : BOOL;
   SSC_Rail_BypassOK : BOOL := 1;
   SSC_Rail_InputsOK : BOOL := 1;
   SSC_RailShuntOK : BOOL;
   SSC_Ready_LT : ALIAS FOR SSC01_Safe3:O.Pt01Data;
   SSC_SafeFlt_OK : BOOL := 1;
   SSC_SafetyIO_OK : BOOL := 1;
   SSC_StdFlt_OK : BOOL := 1;
   SSC_Stop0_OK : BOOL := 1;
   SSC_Stop1_OK : BOOL := 1;
   ST_NoScan_Comment : BOOL;
   STS_Enable_Rail : DINT;
   STS_Rail_Bypass_InputOK : BOOL := 1;
   STS_RCS_PwrDisc_InputOK : BOOL := 1;
   STS_SSC_Safety_NodesOK : BOOL := 1;
   STS_Status_OK : BOOL := 1;
   System_FaultSafeIO : DINT;
   System_FaultSafety : DINT;
   System_FaultStandard : DINT;
   System_Warning : DINT := 134217728;
   Tmr_Rail_Bypass_Disc : TIMER := (PRE := 1000);
   Tmr_Rail_Debn : TIMER := (PRE := 25);
   Tmr_Rail_Shunt : TIMER[7] := ([0].PRE := 2000, [0].ACC := 2000, [0].EN := 1, [0].DN := 1, [1].PRE := 250, [2].PRE := 250, [3].PRE := 250, [4].PRE := 250, [5].PRE := 250, [6].PRE := 250);
   ZZZ_DIAG_A_C1_0302 : BOOL := 1;
   ZZZ_DIAG_A_C2_0302 : BOOL := 1;
   ZZZ_DIAG_A_C3_0302 : BOOL := 1;
   ZZZ_DIAG_C1_AxisFault : DINT := 2;
   ZZZ_DIAG_C1_AxisStatus : DINT;
   ZZZ_DIAG_C1_EnableRail : DINT := 18;
   ZZZ_DIAG_C1_ModuleFault : BOOL;
   ZZZ_DIAG_C1_MotionStatus : DINT;
   ZZZ_DIAG_C1_MSF : MOTION_INSTRUCTION := (FLAGS := 33554432);
   ZZZ_DIAG_C1_MSO : MOTION_INSTRUCTION := (FLAGS := 33554432);
   ZZZ_DIAG_C1_OneTimeOnly : BOOL := 1;
   ZZZ_DIAG_C1_OutputEnable : BOOL;
   ZZZ_DIAG_C1_OutputEnable_ACC : DINT := 29840;
   ZZZ_DIAG_C1_PhysicalAxisFault : BOOL;
   ZZZ_DIAG_C1_ServoActionStatus : BOOL;
   ZZZ_DIAG_C2_AxisFault : DINT := 2;
   ZZZ_DIAG_C2_AxisStatus : DINT;
   ZZZ_DIAG_C2_EnableRail : DINT := 18;
   ZZZ_DIAG_C2_MotionStatus : DINT;
   ZZZ_DIAG_C2_MSF : MOTION_INSTRUCTION := (FLAGS := 33554432);
   ZZZ_DIAG_C2_MSO : MOTION_INSTRUCTION := (FLAGS := 33554432);
   ZZZ_DIAG_C2_OneTimeOnly : BOOL := 1;
   ZZZ_DIAG_C2_OutputEnable : BOOL;
   ZZZ_DIAG_C2_OutputEnable_ACC : DINT := 29839;
   ZZZ_DIAG_C3_AxisFault : DINT := 2;
   ZZZ_DIAG_C3_AxisStatus : DINT;
   ZZZ_DIAG_C3_EnableRail : DINT := 18;
   ZZZ_DIAG_C3_MotionStatus : DINT;
   ZZZ_DIAG_C3_MSF : MOTION_INSTRUCTION := (FLAGS := 33554432);
   ZZZ_DIAG_C3_MSO : MOTION_INSTRUCTION := (FLAGS := 33554432);
   ZZZ_DIAG_C3_OneTimeOnly : BOOL := 1;
   ZZZ_DIAG_C3_OutputEnable : BOOL;
   ZZZ_DIAG_C3_OutputEnable_ACC : DINT := 29839;
   ZZZ_DIAG_ONS : DINT;
   ZZZ_DIAG_S_C1_OutputEnableTON : TIMER := (PRE := 60000, ACC := 60000, EN := 1, DN := 1);
   ZZZ_DIAG_S_C1_SAFETY_ENABLE_1 : BOOL;
   ZZZ_DIAG_S_C1_SAFETY_ENABLE_2 : BOOL;
   ZZZ_DIAG_S_C2_OutputEnableTON : TIMER := (PRE := 60000, ACC := 60009, EN := 1, DN := 1);
   ZZZ_DIAG_S_C2_SAFETY_ENABLE_1 : BOOL;
   ZZZ_DIAG_S_C2_SAFETY_ENABLE_2 : BOOL;
   ZZZ_DIAG_S_C3_OutputEnableTON : TIMER := (PRE := 60000, ACC := 60009, EN := 1, DN := 1);
   ZZZ_DIAG_S_C3_SAFETY_ENABLE_1 : BOOL;
   ZZZ_DIAG_S_C3_SAFETY_ENABLE_2 : BOOL;
END_VAR
